C01840=1102.143,-108.620,-47.409,179.948,4.444,148.747
C01841=1102.137,-108.370,-47.419,179.947,4.449,148.749
C01842=1102.132,-108.121,-47.430,179.947,4.454,148.750
C01843=1102.128,-107.871,-47.440,179.946,4.459,148.751
C01844=1102.122,-107.621,-47.450,179.946,4.464,148.752
C01845=1102.117,-107.371,-47.460,179.946,4.469,148.753
C01846=1102.111,-107.122,-47.471,179.945,4.474,148.755
C01847=1102.106,-106.872,-47.481,179.944,4.479,148.756
C01848=1102.101,-106.622,-47.491,179.944,4.484,148.757
C01849=1102.096,-106.373,-47.501,179.944,4.489,148.758
C01850=1102.091,-106.122,-47.512,179.943,4.494,148.760
C01851=1102.085,-105.873,-47.522,179.943,4.499,148.761
C01852=1102.080,-105.623,-47.532,179.942,4.504,148.762
C01853=1102.075,-105.373,-47.543,179.942,4.509,148.763
C01854=1102.069,-105.124,-47.553,179.941,4.513,148.764
C01855=1102.064,-104.874,-47.564,179.941,4.518,148.766
C01856=1102.059,-104.624,-47.574,179.940,4.524,148.767
C01857=1102.054,-104.375,-47.584,179.940,4.529,148.768
C01858=1102.049,-104.125,-47.594,179.939,4.533,148.769
C01859=1102.043,-103.875,-47.605,179.939,4.539,148.771
C01860=1102.038,-103.625,-47.615,179.939,4.544,148.772
C01861=1102.033,-103.376,-47.625,179.938,4.548,148.773
C01862=1102.028,-103.126,-47.637,179.938,4.553,148.774
C01863=1102.023,-102.876,-47.647,179.938,4.558,148.775
C01864=1102.017,-102.627,-47.657,179.937,4.563,148.777
C01865=1102.012,-102.377,-47.668,179.937,4.568,148.778
C01866=1102.006,-102.127,-47.678,179.936,4.573,148.779
C01867=1102.001,-101.877,-47.689,179.936,4.578,148.780
C01868=1101.997,-101.628,-47.699,179.935,4.583,148.782
C01869=1101.992,-101.378,-47.709,179.935,4.588,148.783
C01870=1101.986,-101.128,-47.720,179.934,4.593,148.784
C01871=1101.981,-100.878,-47.730,179.933,4.597,148.785
C01872=1101.976,-100.664,-47.740,179.933,4.601,148.786
C01873=1101.972,-100.450,-47.748,179.933,4.606,148.787
C01874=1101.967,-100.235,-47.758,179.933,4.611,148.788
C01875=1101.963,-100.022,-47.767,179.932,4.614,148.789
C01876=1101.959,-99.806,-47.776,179.932,4.618,148.790
C01877=1101.954,-99.592,-47.785,179.931,4.623,148.792
C01878=1101.949,-99.378,-47.794,179.931,4.627,148.793
C01879=1101.944,-99.164,-47.803,179.931,4.631,148.793
C01880=1101.939,-98.913,-47.814,179.930,4.636,148.795
C01881=1101.934,-98.664,-47.825,179.930,4.641,148.796
C01882=1101.929,-98.414,-47.835,179.930,4.646,148.797
C01883=1101.923,-98.165,-47.845,179.929,4.651,148.799
C01884=1101.918,-97.914,-47.856,179.929,4.656,148.800
C01885=1101.913,-97.665,-47.867,179.928,4.661,148.801
C01886=1101.908,-97.415,-47.878,179.928,4.665,148.802
C01887=1101.903,-97.166,-47.888,179.927,4.671,148.803
C01888=1101.898,-96.916,-47.899,179.927,4.676,148.805
C01889=1101.892,-96.666,-47.909,179.926,4.680,148.806
C01890=1101.887,-96.416,-47.920,179.926,4.685,148.807
C01891=1101.882,-96.167,-47.931,179.926,4.690,148.808
C01892=1101.877,-95.917,-47.941,179.925,4.695,148.809
C01893=1101.872,-95.668,-47.952,179.925,4.700,148.810
C01894=1101.867,-95.418,-47.963,179.925,4.705,148.812
C01895=1101.862,-95.168,-47.973,179.924,4.709,148.813
C01896=1101.856,-94.919,-47.984,179.924,4.714,148.814
C01897=1101.851,-94.668,-47.995,179.923,4.720,148.815
C01898=1101.845,-94.419,-48.006,179.923,4.725,148.816
C01899=1101.840,-94.169,-48.017,179.922,4.729,148.818
C01900=1101.835,-93.919,-48.027,179.922,4.734,148.819
C01901=1101.830,-93.670,-48.038,179.922,4.739,148.820
C01902=1101.824,-93.420,-48.049,179.921,4.744,148.821
C01903=1101.820,-93.171,-48.060,179.921,4.749,148.822
C01904=1101.815,-92.920,-48.071,179.921,4.754,148.824
C01905=1101.809,-92.671,-48.082,179.921,4.759,148.825
C01906=1101.804,-92.421,-48.093,179.920,4.763,148.826
C01907=1101.798,-92.172,-48.104,179.920,4.769,148.827
C01908=1101.793,-91.922,-48.114,179.919,4.774,148.828
C01909=1101.788,-91.672,-48.125,179.919,4.779,148.830
C01910=1101.783,-91.423,-48.136,179.919,4.783,148.831
C01911=1101.778,-91.172,-48.146,179.918,4.788,148.832
C01912=1101.772,-90.923,-48.158,179.918,4.793,148.833
C01913=1101.767,-90.674,-48.169,179.918,4.799,148.834
C01914=1101.762,-90.423,-48.180,179.918,4.804,148.836
C01915=1101.757,-90.174,-48.191,179.917,4.808,148.837
C01916=1101.752,-89.924,-48.201,179.917,4.813,148.838
C01917=1101.747,-89.674,-48.213,179.917,4.818,148.839
C01918=1101.741,-89.425,-48.223,179.916,4.824,148.840
C01919=1101.736,-89.175,-48.234,179.916,4.829,148.841
C01920=1101.731,-88.925,-48.245,179.916,4.834,148.843
C01921=1101.726,-88.676,-48.256,179.915,4.838,148.844
C01922=1101.721,-88.426,-48.268,179.915,4.844,148.845
C01923=1101.715,-88.176,-48.278,179.914,4.849,148.846
C01924=1101.710,-87.927,-48.289,179.914,4.854,148.848
C01925=1101.705,-87.676,-48.300,179.914,4.859,148.849
C01926=1101.699,-87.427,-48.311,179.914,4.864,148.850
C01927=1101.695,-87.178,-48.323,179.913,4.869,148.851
C01928=1101.691,-86.964,-48.332,179.913,4.873,148.852
C01929=1101.686,-86.749,-48.342,179.913,4.878,148.853
C01930=1101.681,-86.535,-48.351,179.912,4.882,148.854
C01931=1101.677,-86.321,-48.360,179.913,4.886,148.855
C01932=1101.673,-86.106,-48.370,179.912,4.891,148.856
C01933=1101.668,-85.892,-48.380,179.912,4.895,148.857
C01934=1101.664,-85.678,-48.389,179.911,4.900,148.859
C01935=1101.659,-85.463,-48.399,179.911,4.904,148.860
C01936=1101.654,-85.214,-48.409,179.911,4.909,148.861
C01937=1101.649,-84.964,-48.421,179.911,4.914,148.862
C01938=1101.643,-84.714,-48.433,179.911,4.919,148.863
C01939=1101.638,-84.464,-48.443,179.910,4.923,148.864
C01940=1101.633,-84.215,-48.454,179.910,4.929,148.865
C01941=1101.628,-83.965,-48.466,179.909,4.934,148.867
C01942=1101.623,-83.715,-48.477,179.909,4.939,148.868
C01943=1101.617,-83.466,-48.487,179.909,4.944,148.869
C01944=1101.612,-83.216,-48.499,179.909,4.950,148.870
C01945=1101.607,-82.966,-48.511,179.908,4.955,148.872
C01946=1101.603,-82.717,-48.522,179.908,4.960,148.873
C01947=1101.596,-82.467,-48.533,179.908,4.965,148.874
C01948=1101.592,-82.217,-48.544,179.908,4.970,148.875
C01949=1101.586,-81.967,-48.556,179.907,4.974,148.876
C01950=1101.582,-81.718,-48.567,179.907,4.980,148.877
C01951=1101.576,-81.469,-48.578,179.906,4.985,148.879
C01952=1101.570,-81.218,-48.589,179.906,4.990,148.880
C01953=1101.566,-80.968,-48.601,179.906,4.995,148.881
C01954=1101.561,-80.719,-48.612,179.906,5.000,148.882
C01955=1101.555,-80.470,-48.623,179.906,5.006,148.884
C01956=1101.550,-80.220,-48.635,179.905,5.011,148.885
C01957=1101.545,-79.970,-48.647,179.905,5.016,148.886
C01958=1101.540,-79.720,-48.657,179.905,5.021,148.887
C01959=1101.534,-79.471,-48.669,179.905,5.026,148.888
C01960=1101.529,-79.221,-48.680,179.905,5.031,148.890
C01961=1101.524,-78.971,-48.692,179.905,5.036,148.891
C01962=1101.519,-78.721,-48.703,179.903,5.041,148.892
C01963=1101.514,-78.471,-48.715,179.903,5.046,148.893
C01964=1101.508,-78.223,-48.726,179.903,5.051,148.894
C01965=1101.504,-77.973,-48.737,179.903,5.057,148.896
C01966=1101.498,-77.723,-48.749,179.903,5.062,148.897
C01967=1101.493,-77.473,-48.760,179.903,5.067,148.898
C01968=1101.488,-77.223,-48.772,179.902,5.072,148.899
C01969=1101.483,-76.974,-48.782,179.902,5.077,148.900
C01970=1101.477,-76.724,-48.794,179.902,5.082,148.902
C01971=1101.472,-76.474,-48.806,179.902,5.087,148.903
C01972=1101.467,-76.224,-48.818,179.902,5.092,148.904
C01973=1101.462,-75.974,-48.829,179.902,5.098,148.905
C01974=1101.457,-75.725,-48.841,179.902,5.103,148.906
C01975=1101.451,-75.476,-48.852,179.901,5.108,148.907
C01976=1101.446,-75.226,-48.864,179.901,5.113,148.909
C01977=1101.441,-74.976,-48.875,179.901,5.118,148.910
C01978=1101.436,-74.726,-48.887,179.901,5.123,148.911
C01979=1101.431,-74.476,-48.899,179.901,5.128,148.912
C01980=1101.426,-74.227,-48.910,179.901,5.134,148.913
C01981=1101.420,-73.978,-48.921,179.900,5.138,148.914
C01982=1101.414,-73.728,-48.933,179.900,5.143,148.916
C01983=1101.410,-73.479,-48.945,179.900,5.148,148.917
C01984=1101.406,-73.264,-48.955,179.900,5.153,148.918
C01985=1101.401,-73.050,-48.965,179.899,5.157,148.919
C01986=1101.397,-72.835,-48.976,179.900,5.162,148.920
C01987=1101.392,-72.621,-48.985,179.899,5.166,148.921
C01988=1101.389,-72.407,-48.995,179.899,5.170,148.922
C01989=1101.384,-72.193,-49.005,179.899,5.175,148.923
C01990=1101.379,-71.979,-49.015,179.899,5.179,148.924
C01991=1101.375,-71.765,-49.025,179.899,5.183,148.925
C01992=1101.369,-71.515,-49.037,179.898,5.188,148.926
C01993=1101.365,-71.265,-49.049,179.898,5.193,148.927
C01994=1101.359,-71.015,-49.060,179.898,5.198,148.928
C01995=1101.354,-70.765,-49.072,179.898,5.203,148.929
C01996=1101.349,-70.516,-49.084,179.898,5.209,148.931
C01997=1101.343,-70.267,-49.096,179.898,5.214,148.932
C01998=1101.338,-70.017,-49.108,179.898,5.219,148.933
C01999=1101.333,-69.768,-49.119,179.898,5.224,148.934
C02000=1101.328,-69.518,-49.131,179.897,5.229,148.935
C02001=1101.322,-69.268,-49.143,179.898,5.234,148.936
C02002=1101.318,-69.019,-49.155,179.898,5.239,148.937
C02003=1101.312,-68.769,-49.167,179.898,5.244,148.939
C02004=1101.307,-68.519,-49.179,179.897,5.249,148.940
C02005=1101.302,-68.269,-49.190,179.897,5.254,148.941
C02006=1101.297,-68.020,-49.202,179.897,5.259,148.942
C02007=1101.292,-67.770,-49.214,179.897,5.265,148.943
C02008=1101.287,-67.520,-49.226,179.897,5.269,148.944
C02009=1101.282,-67.270,-49.238,179.897,5.274,148.945
C02010=1101.277,-67.021,-49.250,179.897,5.279,148.947
C02011=1101.271,-66.771,-49.262,179.896,5.284,148.948
C02012=1101.266,-66.521,-49.273,179.897,5.289,148.949
C02013=1101.261,-66.272,-49.286,179.897,5.294,148.950
C02014=1101.256,-66.022,-49.298,179.897,5.299,148.951
C02015=1101.250,-65.772,-49.310,179.896,5.304,148.952
C02016=1101.246,-65.523,-49.322,179.897,5.309,148.953
C02017=1101.241,-65.273,-49.334,179.897,5.314,148.954
C02018=1101.235,-65.023,-49.345,179.897,5.319,148.955
C02019=1101.230,-64.774,-49.358,179.896,5.324,148.957
C02020=1101.225,-64.524,-49.370,179.897,5.329,148.958
C02021=1101.220,-64.275,-49.381,179.897,5.334,148.959
C02022=1101.215,-64.025,-49.394,179.897,5.339,148.960
C02023=1101.209,-63.775,-49.406,179.897,5.344,148.961
C02024=1101.204,-63.526,-49.418,179.896,5.348,148.962
C02025=1101.199,-63.276,-49.430,179.897,5.353,148.963
C02026=1101.194,-63.026,-49.442,179.897,5.358,148.964
C02027=1101.189,-62.777,-49.454,179.896,5.363,148.965
C02028=1101.184,-62.527,-49.466,179.897,5.368,148.966
C02029=1101.178,-62.278,-49.479,179.897,5.373,148.967
C02030=1101.173,-62.028,-49.490,179.897,5.378,148.968
C02031=1101.168,-61.779,-49.503,179.897,5.383,148.969
C02032=1101.164,-61.528,-49.515,179.897,5.388,148.970
C02033=1101.159,-61.279,-49.527,179.897,5.393,148.971
C02034=1101.153,-61.029,-49.539,179.897,5.397,148.972
C02035=1101.148,-60.780,-49.552,179.897,5.402,148.974
C02036=1101.143,-60.530,-49.564,179.897,5.407,148.975
C02037=1101.138,-60.280,-49.576,179.897,5.412,148.976
C02038=1101.132,-60.030,-49.588,179.898,5.417,148.977
C02039=1101.127,-59.781,-49.601,179.898,5.422,148.978
C02040=1101.123,-59.567,-49.612,179.897,5.426,148.979
C02041=1101.118,-59.353,-49.621,179.897,5.430,148.980
C02042=1101.114,-59.139,-49.632,179.897,5.433,148.980
C02043=1101.110,-58.924,-49.643,179.898,5.438,148.981
C02044=1101.105,-58.711,-49.653,179.898,5.442,148.982
C02045=1101.101,-58.497,-49.664,179.897,5.446,148.983
C02046=1101.097,-58.282,-49.674,179.897,5.450,148.984
C02047=1101.092,-58.068,-49.684,179.897,5.454,148.985
C02048=1101.087,-57.819,-49.697,179.897,5.459,148.986
C02049=1101.083,-57.569,-49.710,179.897,5.464,148.987
C02050=1101.077,-57.319,-49.721,179.897,5.468,148.988
C02051=1101.072,-57.070,-49.734,179.897,5.473,148.989
C02052=1101.067,-56.820,-49.746,179.897,5.478,148.990
C02053=1101.062,-56.570,-49.759,179.896,5.482,148.991
C02054=1101.056,-56.321,-49.771,179.897,5.487,148.992
C02055=1101.051,-56.071,-49.783,179.897,5.492,148.994
C02056=1101.047,-55.821,-49.796,179.896,5.496,148.994
C02057=1101.041,-55.572,-49.809,179.896,5.501,148.996
C02058=1101.036,-55.322,-49.821,179.896,5.506,148.997
C02059=1101.031,-55.072,-49.833,179.896,5.510,148.998
C02060=1101.026,-54.823,-49.846,179.896,5.515,148.999
C02061=1101.020,-54.573,-49.858,179.896,5.520,149.000
C02062=1101.016,-54.323,-49.871,179.896,5.525,149.001
C02063=1101.011,-54.074,-49.883,179.896,5.529,149.002
C02064=1101.006,-53.825,-49.896,179.896,5.534,149.003
C02065=1101.000,-53.575,-49.908,179.896,5.539,149.004
C02066=1100.995,-53.325,-49.920,179.895,5.544,149.005
C02067=1100.990,-53.075,-49.933,179.896,5.548,149.006
C02068=1100.985,-52.826,-49.946,179.896,5.553,149.007
C02069=1100.980,-52.576,-49.958,179.895,5.558,149.009
C02070=1100.974,-52.326,-49.971,179.895,5.562,149.009
C02071=1100.969,-52.077,-49.983,179.895,5.568,149.011
C02072=1100.964,-51.827,-49.996,179.894,5.572,149.012
C02073=1100.959,-51.577,-50.008,179.895,5.577,149.013
C02074=1100.954,-51.328,-50.021,179.895,5.582,149.014
C02075=1100.949,-51.078,-50.034,179.894,5.586,149.015
C02076=1100.944,-50.828,-50.047,179.895,5.591,149.016
C02077=1100.939,-50.579,-50.059,179.894,5.596,149.017
C02078=1100.934,-50.329,-50.071,179.894,5.600,149.018
C02079=1100.929,-50.080,-50.084,179.894,5.605,149.019
C02080=1100.923,-49.830,-50.097,179.894,5.610,149.020
C02081=1100.918,-49.580,-50.110,179.893,5.614,149.022
C02082=1100.913,-49.331,-50.122,179.894,5.619,149.022
C02083=1100.908,-49.082,-50.135,179.894,5.624,149.024
C02084=1100.903,-48.832,-50.148,179.893,5.629,149.025
C02085=1100.898,-48.582,-50.160,179.894,5.633,149.026
C02086=1100.893,-48.332,-50.172,179.893,5.638,149.027
C02087=1100.887,-48.083,-50.186,179.893,5.643,149.028
C02088=1100.882,-47.833,-50.199,179.893,5.647,149.029
C02089=1100.877,-47.583,-50.211,179.893,5.652,149.030
C02090=1100.872,-47.334,-50.224,179.893,5.657,149.031
C02091=1100.867,-47.085,-50.236,179.892,5.662,149.032
C02092=1100.862,-46.834,-50.250,179.892,5.666,149.033
C02093=1100.857,-46.585,-50.263,179.892,5.671,149.034
C02094=1100.852,-46.336,-50.275,179.892,5.676,149.036
C02095=1100.847,-46.086,-50.288,179.892,5.680,149.036
C02096=1100.842,-45.872,-50.298,179.891,5.684,149.038
C02097=1100.838,-45.658,-50.310,179.892,5.689,149.039
C02098=1100.834,-45.443,-50.321,179.892,5.693,149.039
C02099=1100.829,-45.229,-50.333,179.891,5.697,149.040
C02100=1100.824,-45.016,-50.343,179.891,5.701,149.041
C02101=1100.820,-44.802,-50.354,179.891,5.705,149.042
C02102=1100.816,-44.587,-50.365,179.891,5.709,149.043
C02103=1100.812,-44.374,-50.376,179.891,5.713,149.044
C02104=1100.807,-44.124,-50.389,179.891,5.718,149.045
C02105=1100.801,-43.875,-50.402,179.891,5.723,149.046
C02106=1100.796,-43.625,-50.415,179.890,5.727,149.047
C02107=1100.791,-43.375,-50.428,179.890,5.732,149.048
C02108=1100.786,-43.126,-50.440,179.890,5.736,149.050
C02109=1100.781,-42.876,-50.454,179.890,5.741,149.051
C02110=1100.776,-42.626,-50.466,179.890,5.746,149.052
C02111=1100.771,-42.377,-50.479,179.889,5.751,149.053
C02112=1100.766,-42.127,-50.492,179.889,5.756,149.054
C02113=1100.760,-41.877,-50.505,179.890,5.760,149.055
C02114=1100.756,-41.627,-50.518,179.889,5.765,149.056
C02115=1100.751,-41.378,-50.531,179.890,5.769,149.057
C02116=1100.745,-41.128,-50.544,179.889,5.774,149.058
C02117=1100.740,-40.878,-50.557,179.889,5.779,149.059
C02118=1100.735,-40.630,-50.570,179.889,5.783,149.060
C02119=1100.730,-40.380,-50.583,179.889,5.788,149.061
C02120=1100.725,-40.130,-50.596,179.889,5.793,149.062
C02121=1100.720,-39.881,-50.609,179.889,5.797,149.063
C02122=1100.715,-39.630,-50.623,179.889,5.802,149.064
C02123=1100.710,-39.381,-50.635,179.889,5.806,149.065
C02124=1100.704,-39.131,-50.648,179.889,5.810,149.066
C02125=1100.700,-38.882,-50.662,179.889,5.816,149.067
C02126=1100.694,-38.633,-50.675,179.889,5.819,149.068
C02127=1100.689,-38.382,-50.688,179.889,5.824,149.069
C02128=1100.684,-38.133,-50.701,179.889,5.828,149.070
C02129=1100.679,-37.884,-50.713,179.890,5.833,149.071
C02130=1100.674,-37.634,-50.728,179.890,5.838,149.072
C02131=1100.669,-37.385,-50.740,179.890,5.842,149.073
C02132=1100.664,-37.134,-50.754,179.890,5.847,149.074
C02133=1100.658,-36.885,-50.767,179.890,5.851,149.075
C02134=1100.654,-36.636,-50.780,179.890,5.855,149.076
C02135=1100.648,-36.386,-50.793,179.890,5.859,149.077
C02136=1100.643,-36.137,-50.806,179.891,5.864,149.078
C02137=1100.638,-35.886,-50.820,179.891,5.869,149.078
C02138=1100.633,-35.638,-50.833,179.891,5.873,149.079
C02139=1100.628,-35.387,-50.846,179.891,5.877,149.080
C02140=1100.623,-35.138,-50.859,179.892,5.882,149.081
C02141=1100.618,-34.888,-50.873,179.892,5.886,149.082
C02142=1100.613,-34.639,-50.886,179.892,5.891,149.083
C02143=1100.607,-34.389,-50.899,179.892,5.895,149.084
C02144=1100.603,-34.140,-50.913,179.892,5.899,149.085
C02145=1100.598,-33.890,-50.926,179.893,5.904,149.086
C02146=1100.592,-33.640,-50.939,179.893,5.908,149.087
C02147=1100.588,-33.391,-50.953,179.893,5.913,149.088
C02148=1100.582,-33.141,-50.966,179.894,5.918,149.088
C02149=1100.578,-32.891,-50.979,179.893,5.921,149.089
C02150=1100.572,-32.642,-50.993,179.894,5.926,149.090
C02151=1100.568,-32.392,-51.006,179.895,5.931,149.091
C02152=1100.559,-32.014,-51.027,179.895,5.937,149.092
C02153=1100.552,-31.636,-51.047,179.896,5.944,149.094
C02154=1100.544,-31.258,-51.067,179.896,5.951,149.095
C02155=1100.536,-30.879,-51.087,179.896,5.957,149.096
C02156=1100.531,-30.629,-51.101,179.897,5.962,149.097
C02157=1100.526,-30.380,-51.114,179.897,5.967,149.098
C02158=1100.521,-30.130,-51.128,179.898,5.971,149.099
C02159=1100.515,-29.881,-51.141,179.898,5.975,149.100
C02160=1100.511,-29.631,-51.155,179.899,5.980,149.101
C02161=1100.505,-29.382,-51.168,179.899,5.984,149.102
C02162=1100.501,-29.132,-51.182,179.900,5.989,149.103
C02163=1100.495,-28.883,-51.195,179.900,5.994,149.103
C02164=1100.490,-28.633,-51.209,179.900,5.999,149.104
C02165=1100.486,-28.383,-51.222,179.900,6.003,149.105
C02166=1100.480,-28.134,-51.236,179.901,6.007,149.106
C02167=1100.476,-27.884,-51.249,179.901,6.012,149.107
C02168=1100.470,-27.635,-51.263,179.902,6.017,149.108
C02169=1100.465,-27.385,-51.277,179.902,6.021,149.109
C02170=1100.461,-27.135,-51.290,179.903,6.026,149.110
C02171=1100.455,-26.886,-51.304,179.903,6.031,149.111
C02172=1100.450,-26.636,-51.318,179.904,6.036,149.112
C02173=1100.445,-26.387,-51.331,179.904,6.040,149.113
C02174=1100.440,-26.138,-51.345,179.905,6.045,149.113
C02175=1100.435,-25.887,-51.359,179.905,6.050,149.114
C02176=1100.430,-25.638,-51.372,179.905,6.055,149.115
C02177=1100.425,-25.388,-51.386,179.906,6.059,149.116
C02178=1100.419,-25.139,-51.400,179.906,6.064,149.117
C02179=1100.415,-24.890,-51.413,179.906,6.068,149.118
C02180=1100.188,-34.518,-50.930,179.897,5.896,149.083
C02181=1100.194,-34.768,-50.916,179.897,5.892,149.082
C02182=1100.199,-35.018,-50.904,179.897,5.887,149.081
C02183=1100.204,-35.267,-50.890,179.897,5.882,149.080
C02184=1100.209,-35.517,-50.877,179.897,5.878,149.079
C02185=1100.214,-35.766,-50.864,179.896,5.874,149.078
C02186=1100.219,-36.016,-50.851,179.896,5.870,149.077
C02187=1100.224,-36.265,-50.837,179.896,5.865,149.076
C02188=1100.229,-36.515,-50.824,179.895,5.860,149.075
C02189=1100.234,-36.765,-50.811,179.896,5.856,149.074
C02190=1100.239,-37.014,-50.797,179.895,5.851,149.073
C02191=1100.244,-37.264,-50.784,179.895,5.848,149.072
C02192=1100.250,-37.514,-50.771,179.895,5.842,149.071
C02193=1100.255,-37.763,-50.758,179.896,5.838,149.070
C02194=1100.260,-38.012,-50.745,179.895,5.834,149.070
C02195=1100.265,-38.262,-50.731,179.895,5.829,149.069
C02196=1100.270,-38.512,-50.719,179.895,5.825,149.068
C02197=1100.275,-38.762,-50.705,179.895,5.820,149.067
C02198=1100.280,-39.011,-50.692,179.895,5.816,149.066
C02199=1100.285,-39.261,-50.679,179.895,5.811,149.065
C02200=1100.291,-39.510,-50.666,179.895,5.807,149.064
C02201=1100.296,-39.760,-50.653,179.895,5.802,149.063
C02202=1100.300,-40.010,-50.640,179.895,5.798,149.062
C02203=1100.306,-40.259,-50.627,179.895,5.793,149.061
C02204=1100.310,-40.509,-50.613,179.895,5.788,149.060
C02205=1100.316,-40.758,-50.600,179.895,5.784,149.059
C02206=1100.321,-41.008,-50.587,179.895,5.779,149.058
C02207=1100.326,-41.258,-50.574,179.895,5.775,149.056
C02208=1100.332,-41.507,-50.561,179.895,5.770,149.056
C02209=1100.337,-41.757,-50.549,179.896,5.766,149.054
C02210=1100.341,-42.007,-50.536,179.896,5.761,149.053
C02211=1100.347,-42.256,-50.522,179.895,5.756,149.052
C02212=1100.351,-42.506,-50.509,179.896,5.752,149.051
C02213=1100.356,-42.755,-50.496,179.896,5.747,149.050
C02214=1100.362,-43.004,-50.484,179.897,5.742,149.049
C02215=1100.367,-43.255,-50.470,179.896,5.738,149.048
C02216=1100.372,-43.504,-50.457,179.896,5.733,149.047
C02217=1100.377,-43.753,-50.445,179.897,5.728,149.046
C02218=1100.382,-44.004,-50.431,179.897,5.723,149.045
C02219=1100.387,-44.253,-50.419,179.896,5.718,149.044
C02220=1100.393,-44.502,-50.406,179.897,5.714,149.042
C02221=1100.400,-44.896,-50.386,179.897,5.706,149.041
C02222=1100.409,-45.290,-50.365,179.897,5.699,149.039
C02223=1100.416,-45.684,-50.345,179.898,5.692,149.037
C02224=1100.424,-46.077,-50.325,179.898,5.684,149.036
C02225=1100.430,-46.327,-50.312,179.898,5.679,149.034
C02226=1100.435,-46.577,-50.299,179.898,5.675,149.033
C02227=1100.440,-46.826,-50.286,179.898,5.670,149.032
C02228=1100.445,-47.076,-50.273,179.898,5.665,149.031
C02229=1100.450,-47.326,-50.260,179.899,5.661,149.030
C02230=1100.455,-47.575,-50.247,179.899,5.656,149.029
C02231=1100.460,-47.825,-50.235,179.899,5.651,149.028
C02232=1100.466,-48.075,-50.223,179.899,5.646,149.027
C02233=1100.470,-48.325,-50.210,179.899,5.642,149.026
C02234=1100.475,-48.574,-50.197,179.899,5.637,149.025
C02235=1100.481,-48.824,-50.184,179.900,5.632,149.024
C02236=1100.486,-49.074,-50.171,179.899,5.628,149.023
C02237=1100.491,-49.323,-50.158,179.899,5.622,149.021
C02238=1100.496,-49.572,-50.146,179.900,5.618,149.020
C02239=1100.501,-49.822,-50.133,179.900,5.613,149.019
C02240=1100.506,-50.072,-50.120,179.900,5.608,149.018
C02241=1100.512,-50.322,-50.108,179.900,5.604,149.017
C02242=1100.517,-50.571,-50.095,179.901,5.599,149.016
C02243=1100.522,-50.821,-50.083,179.900,5.594,149.015
C02244=1100.527,-51.071,-50.070,179.901,5.590,149.014
C02245=1100.532,-51.320,-50.057,179.901,5.585,149.013
C02246=1100.537,-51.569,-50.044,179.900,5.580,149.012
C02247=1100.542,-51.819,-50.033,179.901,5.576,149.011
C02248=1100.547,-52.068,-50.020,179.901,5.570,149.009
C02249=1100.552,-52.318,-50.007,179.901,5.566,149.009
C02250=1100.558,-52.568,-49.994,179.901,5.561,149.007
C02251=1100.563,-52.817,-49.981,179.902,5.556,149.006
C02252=1100.568,-53.067,-49.969,179.901,5.552,149.005
C02253=1100.573,-53.317,-49.956,179.902,5.547,149.004
C02254=1100.578,-53.567,-49.944,179.901,5.542,149.003
C02255=1100.583,-53.816,-49.931,179.901,5.537,149.002
C02256=1100.589,-54.066,-49.919,179.902,5.533,149.001
C02257=1100.594,-54.315,-49.907,179.902,5.528,149.000
C02258=1100.598,-54.565,-49.894,179.902,5.523,148.999
C02259=1100.603,-54.815,-49.881,179.903,5.519,148.998
C02260=1100.609,-55.064,-49.869,179.902,5.514,148.997
C02261=1100.614,-55.314,-49.857,179.902,5.509,148.996
C02262=1100.619,-55.563,-49.844,179.902,5.505,148.995
C02263=1100.624,-55.814,-49.832,179.903,5.500,148.994
C02264=1100.629,-56.063,-49.819,179.903,5.495,148.992
C02265=1100.634,-56.312,-49.807,179.903,5.491,148.991
C02266=1100.640,-56.562,-49.795,179.903,5.486,148.990
C02267=1100.645,-56.812,-49.782,179.902,5.481,148.989
C02268=1100.650,-57.061,-49.769,179.903,5.476,148.988
C02269=1100.655,-57.312,-49.757,179.903,5.472,148.987
C02270=1100.660,-57.561,-49.745,179.903,5.467,148.986
C02271=1100.665,-57.810,-49.732,179.903,5.462,148.985
C02272=1100.670,-58.060,-49.720,179.903,5.458,148.984
C02273=1100.674,-58.274,-49.709,179.903,5.454,148.983
C02274=1100.679,-58.488,-49.699,179.903,5.449,148.982
C02275=1100.683,-58.702,-49.688,179.903,5.445,148.981
C02276=1100.687,-58.916,-49.678,179.903,5.441,148.980
C02277=1100.692,-59.130,-49.667,179.904,5.437,148.979
C02278=1100.696,-59.345,-49.656,179.904,5.433,148.978
C02279=1100.701,-59.559,-49.646,179.904,5.429,148.978
C02280=1100.705,-59.773,-49.636,179.904,5.425,148.977
C02281=1100.710,-60.022,-49.623,179.903,5.420,148.976
C02282=1100.716,-60.272,-49.611,179.904,5.416,148.974
C02283=1100.721,-60.521,-49.599,179.903,5.411,148.974
C02284=1100.726,-60.771,-49.587,179.904,5.406,148.972
C02285=1100.730,-61.021,-49.574,179.903,5.401,148.971
C02286=1100.736,-61.271,-49.562,179.903,5.396,148.970
C02287=1100.741,-61.520,-49.550,179.903,5.391,148.969
C02288=1100.746,-61.770,-49.538,179.903,5.386,148.968
C02289=1100.751,-62.020,-49.525,179.903,5.381,148.967
C02290=1100.757,-62.270,-49.513,179.903,5.377,148.966
C02291=1100.762,-62.519,-49.501,179.903,5.372,148.965
C02292=1100.767,-62.768,-49.490,179.903,5.367,148.964
C02293=1100.772,-63.018,-49.477,179.903,5.362,148.963
C02294=1100.777,-63.268,-49.465,179.903,5.357,148.962
C02295=1100.782,-63.517,-49.452,179.903,5.352,148.961
C02296=1100.788,-63.767,-49.441,179.903,5.347,148.960
C02297=1100.793,-64.016,-49.428,179.903,5.342,148.959
C02298=1100.798,-64.266,-49.417,179.903,5.337,148.957
C02299=1100.803,-64.516,-49.405,179.903,5.333,148.957
C02300=1100.807,-64.766,-49.392,179.903,5.328,148.955
C02301=1100.813,-65.016,-49.380,179.903,5.323,148.954
C02302=1100.818,-65.265,-49.367,179.903,5.318,148.953
C02303=1100.823,-65.515,-49.356,179.903,5.313,148.952
C02304=1100.828,-65.765,-49.344,179.903,5.308,148.951
C02305=1100.833,-66.014,-49.332,179.903,5.303,148.950
C02306=1100.839,-66.264,-49.320,179.903,5.298,148.949
C02307=1100.843,-66.514,-49.308,179.903,5.293,148.948
C02308=1100.849,-66.763,-49.296,179.903,5.288,148.947
C02309=1100.854,-67.013,-49.284,179.903,5.283,148.945
C02310=1100.859,-67.263,-49.272,179.903,5.277,148.944
C02311=1100.864,-67.512,-49.260,179.903,5.273,148.943
C02312=1100.869,-67.762,-49.248,179.904,5.268,148.942
C02313=1100.875,-68.012,-49.236,179.904,5.263,148.941
C02314=1100.880,-68.262,-49.224,179.904,5.258,148.940
C02315=1100.884,-68.511,-49.212,179.904,5.253,148.939
C02316=1100.890,-68.761,-49.200,179.904,5.248,148.937
C02317=1100.896,-69.010,-49.189,179.904,5.243,148.936
C02318=1100.901,-69.259,-49.178,179.904,5.238,148.935
C02319=1100.906,-69.509,-49.165,179.904,5.233,148.934
C02320=1100.911,-69.759,-49.153,179.904,5.228,148.933
C02321=1100.917,-70.009,-49.141,179.904,5.223,148.932
C02322=1100.921,-70.258,-49.130,179.904,5.217,148.931
C02323=1100.927,-70.508,-49.118,179.905,5.212,148.929
C02324=1100.932,-70.757,-49.105,179.905,5.207,148.928
C02325=1100.937,-71.007,-49.094,179.905,5.202,148.927
C02326=1100.942,-71.257,-49.082,179.905,5.197,148.926
C02327=1100.947,-71.507,-49.070,179.905,5.192,148.925
C02328=1100.952,-71.757,-49.059,179.905,5.187,148.924
C02329=1100.957,-71.970,-49.049,179.905,5.183,148.923
C02330=1100.961,-72.185,-49.039,179.906,5.179,148.922
C02331=1100.966,-72.399,-49.028,179.905,5.174,148.921
C02332=1100.970,-72.613,-49.018,179.906,5.170,148.920
C02333=1100.975,-72.827,-49.008,179.906,5.166,148.919
C02334=1100.978,-73.041,-48.999,179.906,5.161,148.918
C02335=1100.983,-73.256,-48.989,179.906,5.157,148.917
C02336=1100.987,-73.470,-48.978,179.906,5.152,148.916
C02337=1100.993,-73.719,-48.967,179.906,5.147,148.914
C02338=1100.998,-73.969,-48.955,179.907,5.142,148.913
C02339=1101.003,-74.219,-48.944,179.907,5.137,148.912
C02340=1101.009,-74.469,-48.932,179.907,5.132,148.911
C02341=1101.013,-74.718,-48.920,179.908,5.127,148.910
C02342=1101.019,-74.968,-48.909,179.908,5.122,148.909
C02343=1101.024,-75.218,-48.897,179.908,5.117,148.907
C02344=1101.030,-75.467,-48.886,179.908,5.112,148.906
C02345=1101.034,-75.717,-48.874,179.908,5.107,148.905
C02346=1101.040,-75.967,-48.863,179.908,5.101,148.904
C02347=1101.044,-76.216,-48.851,179.908,5.096,148.903
C02348=1101.050,-76.466,-48.839,179.909,5.091,148.902
C02349=1101.055,-76.716,-48.827,179.909,5.086,148.900
C02350=1101.060,-76.966,-48.816,179.909,5.081,148.899
C02351=1101.066,-77.215,-48.805,179.909,5.076,148.898
C02352=1101.071,-77.465,-48.793,179.909,5.071,148.897
C02353=1101.076,-77.715,-48.781,179.909,5.065,148.896
C02354=1101.081,-77.964,-48.770,179.910,5.060,148.894
C02355=1101.086,-78.214,-48.758,179.910,5.055,148.893
C02356=1101.092,-78.463,-48.747,179.910,5.051,148.892
C02357=1101.097,-78.713,-48.736,179.911,5.046,148.891
C02358=1101.102,-78.963,-48.724,179.911,5.041,148.890
C02359=1101.107,-79.212,-48.712,179.911,5.035,148.888
C02360=1101.112,-79.462,-48.701,179.912,5.030,148.887
C02361=1101.117,-79.711,-48.690,179.912,5.025,148.886
C02362=1101.123,-79.961,-48.678,179.912,5.020,148.885
C02363=1101.128,-80.211,-48.668,179.912,5.014,148.884
C02364=1101.133,-80.461,-48.656,179.912,5.009,148.882
C02365=1101.138,-80.711,-48.644,179.912,5.004,148.881
C02366=1101.144,-80.960,-48.633,179.913,4.999,148.880
C02367=1101.148,-81.210,-48.622,179.913,4.994,148.879
C02368=1101.154,-81.460,-48.610,179.913,4.989,148.878
C02369=1101.158,-81.709,-48.599,179.914,4.984,148.876
C02370=1101.164,-81.959,-48.588,179.914,4.979,148.875
C02371=1101.170,-82.209,-48.576,179.914,4.974,148.874
C02372=1101.174,-82.458,-48.565,179.915,4.969,148.873
C02373=1101.180,-82.708,-48.553,179.915,4.964,148.872
C02374=1101.185,-82.957,-48.542,179.915,4.958,148.870
C02375=1101.190,-83.207,-48.532,179.915,4.953,148.869
C02376=1101.195,-83.457,-48.520,179.915,4.948,148.868
C02377=1101.200,-83.707,-48.509,179.915,4.943,148.867
C02378=1101.205,-83.956,-48.498,179.916,4.938,148.866
C02379=1101.211,-84.206,-48.486,179.916,4.932,148.864
C02380=1101.216,-84.456,-48.475,179.917,4.928,148.863
C02381=1101.221,-84.705,-48.464,179.917,4.923,148.862
C02382=1101.226,-84.955,-48.452,179.917,4.918,148.861
C02383=1101.231,-85.205,-48.442,179.918,4.913,148.859
C02384=1101.236,-85.455,-48.431,179.918,4.907,148.858
C02385=1101.241,-85.669,-48.421,179.918,4.904,148.857
C02386=1101.246,-85.883,-48.411,179.918,4.898,148.856
C02387=1101.250,-86.098,-48.402,179.919,4.894,148.855
C02388=1101.255,-86.312,-48.392,179.919,4.890,148.854
C02389=1101.259,-86.526,-48.383,179.919,4.885,148.853
C02390=1101.263,-86.741,-48.373,179.919,4.881,148.852
C02391=1101.268,-86.955,-48.363,179.920,4.877,148.851
C02392=1101.272,-87.169,-48.354,179.920,4.872,148.850
C02393=1101.278,-87.418,-48.343,179.920,4.868,148.849
C02394=1101.282,-87.668,-48.331,179.921,4.863,148.848
C02395=1101.288,-87.918,-48.321,179.921,4.858,148.846
C02396=1101.293,-88.167,-48.310,179.921,4.853,148.845
C02397=1101.298,-88.417,-48.298,179.921,4.847,148.844
C02398=1101.304,-88.667,-48.288,179.921,4.842,148.843
C02399=1101.308,-88.916,-48.276,179.923,4.838,148.841
C02400=1101.313,-89.167,-48.266,179.923,4.832,148.840
C02401=1101.319,-89.416,-48.254,179.923,4.827,148.839
C02402=1101.324,-89.665,-48.243,179.923,4.822,148.838
C02403=1101.329,-89.916,-48.232,179.923,4.817,148.837
C02404=1101.334,-90.165,-48.222,179.924,4.812,148.836
C02405=1101.339,-90.415,-48.211,179.924,4.808,148.834
C02406=1101.345,-90.664,-48.199,179.925,4.802,148.833
C02407=1101.350,-90.914,-48.189,179.925,4.797,148.832
C02408=1101.355,-91.164,-48.178,179.925,4.792,148.831
C02409=1101.361,-91.414,-48.167,179.925,4.787,148.830
C02410=1101.365,-91.663,-48.156,179.926,4.783,148.828
C02411=1101.371,-91.914,-48.145,179.926,4.777,148.827
C02412=1101.376,-92.163,-48.134,179.926,4.772,148.826
C02413=1101.381,-92.413,-48.123,179.927,4.767,148.825
C02414=1101.387,-92.662,-48.112,179.927,4.763,148.824
C02415=1101.392,-92.912,-48.102,179.927,4.758,148.822
C02416=1101.396,-93.162,-48.091,179.928,4.753,148.821
C02417=1101.402,-93.411,-48.080,179.928,4.747,148.820
C02418=1101.407,-93.661,-48.068,179.929,4.743,148.819
C02419=1101.413,-93.911,-48.058,179.929,4.738,148.818
C02420=1101.418,-94.160,-48.047,179.929,4.733,148.816
C02421=1101.423,-94.410,-48.037,179.929,4.728,148.815
C02422=1101.428,-94.659,-48.025,179.930,4.723,148.814
C02423=1101.433,-94.910,-48.015,179.930,4.718,148.813
C02424=1101.439,-95.159,-48.005,179.930,4.713,148.812
C02425=1101.443,-95.409,-47.993,179.931,4.709,148.810
C02426=1101.450,-95.659,-47.983,179.931,4.704,148.809
C02427=1101.454,-95.908,-47.971,179.932,4.698,148.808
C02428=1101.460,-96.158,-47.961,179.932,4.694,148.807
C02429=1101.465,-96.408,-47.951,179.933,4.689,148.806
C02430=1101.470,-96.657,-47.940,179.933,4.684,148.804
C02431=1101.475,-96.907,-47.929,179.934,4.680,148.803
C02432=1101.480,-97.157,-47.918,179.934,4.674,148.802
C02433=1101.486,-97.407,-47.908,179.934,4.669,148.801
C02434=1101.491,-97.657,-47.897,179.935,4.665,148.800
C02435=1101.496,-97.906,-47.886,179.935,4.660,148.799
C02436=1101.501,-98.156,-47.875,179.935,4.655,148.797
C02437=1101.506,-98.405,-47.865,179.936,4.650,148.796
C02438=1101.511,-98.655,-47.854,179.936,4.645,148.795
C02439=1101.517,-98.905,-47.844,179.937,4.640,148.794
C02440=1101.522,-99.155,-47.833,179.937,4.636,148.793
C02441=1101.527,-99.369,-47.824,179.938,4.631,148.791
C02442=1101.531,-99.584,-47.815,179.938,4.627,148.790
C02443=1101.536,-99.798,-47.806,179.938,4.623,148.789
C02444=1101.540,-100.011,-47.797,179.939,4.618,148.788
C02445=1101.544,-100.227,-47.788,179.939,4.614,148.787
C02446=1101.549,-100.441,-47.778,179.940,4.610,148.786
C02447=1101.553,-100.655,-47.769,179.940,4.605,148.785
C02448=1101.559,-100.869,-47.760,179.940,4.601,148.784
C02449=1101.564,-101.120,-47.750,179.941,4.597,148.783
C02450=1101.569,-101.369,-47.739,179.941,4.592,148.782
C02451=1101.574,-101.619,-47.728,179.941,4.587,148.781
C02452=1101.579,-101.868,-47.718,179.942,4.582,148.779
C02453=1101.584,-102.119,-47.707,179.943,4.577,148.778
C02454=1101.589,-102.367,-47.697,179.943,4.572,148.777
C02455=1101.594,-102.618,-47.686,179.943,4.566,148.775
C02456=1101.600,-102.867,-47.676,179.944,4.562,148.774
C02457=1101.605,-103.117,-47.666,179.944,4.557,148.773
C02458=1101.610,-103.367,-47.655,179.945,4.552,148.772
C02459=1101.615,-103.616,-47.645,179.945,4.548,148.771
C02460=1101.620,-103.866,-47.634,179.946,4.542,148.769
C02461=1101.626,-104.116,-47.624,179.946,4.537,148.768
C02462=1101.631,-104.366,-47.613,179.947,4.533,148.767
C02463=1101.637,-104.615,-47.603,179.947,4.528,148.766
C02464=1101.642,-104.866,-47.592,179.948,4.522,148.764
C02465=1101.647,-105.115,-47.582,179.948,4.517,148.763
C02466=1101.652,-105.364,-47.572,179.949,4.513,148.762
C02467=1101.657,-105.614,-47.561,179.949,4.508,148.761
C02468=1101.662,-105.864,-47.551,179.949,4.502,148.760
C02469=1101.667,-106.114,-47.541,179.950,4.498,148.758
C02470=1101.673,-106.363,-47.530,179.950,4.493,148.757
C02471=1101.679,-106.613,-47.520,179.951,4.488,148.756
C02472=1101.684,-106.863,-47.510,179.951,4.483,148.755
C02473=1101.689,-107.113,-47.499,179.952,4.478,148.753
C02474=1101.693,-107.363,-47.489,179.952,4.473,148.752
C02475=1101.699,-107.612,-47.479,179.953,4.468,148.751
C02476=1101.705,-107.862,-47.469,179.953,4.463,148.750
C02477=1101.710,-108.112,-47.458,179.954,4.458,148.749
C02478=1101.715,-108.361,-47.448,179.954,4.453,148.747
C02479=1101.720,-108.611,-47.437,179.955,4.448,148.746
C02480=1101.725,-108.860,-47.427,179.955,4.443,148.745
C02481=1101.730,-109.110,-47.417,179.956,4.438,148.743
C02482=1101.735,-109.360,-47.406,179.956,4.433,148.742
C02483=1101.741,-109.610,-47.396,179.956,4.428,148.741
C02484=1101.747,-109.859,-47.386,179.957,4.423,148.740
C02485=1101.751,-110.109,-47.376,179.958,4.418,148.738
C02486=1101.756,-110.359,-47.366,179.958,4.413,148.737
C02487=1101.762,-110.609,-47.356,179.958,4.408,148.736
C02488=1101.767,-110.859,-47.346,179.959,4.403,148.735
C02489=1101.773,-111.109,-47.336,179.959,4.398,148.734
C02490=1101.778,-111.358,-47.326,179.960,4.393,148.732
C02491=1101.783,-111.608,-47.315,179.960,4.387,148.731
C02492=1101.788,-111.858,-47.305,179.961,4.383,148.730
C02493=1101.794,-112.107,-47.295,179.962,4.378,148.728
C02494=1101.798,-112.357,-47.285,179.962,4.373,148.727
C02495=1101.804,-112.607,-47.275,179.963,4.367,148.726
C02496=1101.809,-112.856,-47.265,179.963,4.363,148.725
C02497=1101.814,-113.071,-47.256,179.963,4.358,148.724
C02498=1101.818,-113.286,-47.248,179.964,4.354,148.722
C02499=1101.822,-113.500,-47.239,179.964,4.350,148.721
C02500=1101.827,-113.714,-47.230,179.965,4.346,148.720
C02501=1101.832,-113.929,-47.221,179.965,4.341,148.719
C02502=1101.836,-114.143,-47.213,179.966,4.336,148.718
C02503=1101.841,-114.357,-47.204,179.966,4.332,148.717
C02504=1101.845,-114.572,-47.196,179.967,4.328,148.716
C02505=1101.851,-114.821,-47.185,179.967,4.323,148.715
C02506=1101.856,-115.071,-47.175,179.968,4.317,148.713
C02507=1101.861,-115.321,-47.166,179.968,4.312,148.712
C02508=1101.866,-115.571,-47.156,179.969,4.308,148.711
C02509=1101.872,-115.820,-47.145,179.969,4.303,148.710
C02510=1101.876,-116.070,-47.135,179.970,4.297,148.708
C02511=1101.882,-116.320,-47.125,179.970,4.292,148.707
C02512=1101.887,-116.569,-47.115,179.971,4.287,148.706
C02513=1101.893,-116.819,-47.106,179.972,4.282,148.704
C02514=1101.898,-117.070,-47.096,179.972,4.277,148.703
C02515=1101.903,-117.319,-47.085,179.973,4.272,148.702
C02516=1101.908,-117.568,-47.076,179.973,4.266,148.700
C02517=1101.914,-117.818,-47.066,179.974,4.261,148.699
C02518=1101.919,-118.069,-47.056,179.974,4.256,148.698
C02519=1101.924,-118.318,-47.046,179.975,4.251,148.696
C02520=1101.929,-118.567,-47.036,179.976,4.246,148.695
C02521=1101.935,-118.818,-47.026,179.976,4.241,148.694
C02522=1101.940,-119.068,-47.016,179.977,4.236,148.692
C02523=1101.945,-119.317,-47.006,179.977,4.230,148.691
C02524=1101.950,-119.566,-46.997,179.978,4.226,148.690
C02525=1101.956,-119.817,-46.987,179.979,4.221,148.689
C02526=1101.962,-120.066,-46.977,179.979,4.215,148.687
C02527=1101.966,-120.316,-46.967,179.980,4.210,148.686
C02528=1101.972,-120.566,-46.957,179.980,4.205,148.685
C02529=1101.977,-120.815,-46.948,179.981,4.199,148.683
C02530=1101.982,-121.065,-46.938,179.981,4.194,148.682
C02531=1101.987,-121.315,-46.929,179.982,4.190,148.681
C02532=1101.992,-121.565,-46.918,179.983,4.184,148.679
C02533=1101.997,-121.814,-46.909,179.983,4.179,148.678
C02534=1102.003,-122.064,-46.899,179.984,4.173,148.677
C02535=1102.009,-122.314,-46.889,179.984,4.168,148.675
C02536=1102.014,-122.564,-46.880,179.985,4.163,148.674
C02537=1102.019,-122.814,-46.869,179.985,4.158,148.673
C02538=1102.024,-123.063,-46.860,179.986,4.153,148.671
C02539=1102.030,-123.313,-46.850,179.987,4.148,148.670
C02540=1102.035,-123.563,-46.841,179.988,4.142,148.669
C02541=1102.040,-123.812,-46.830,179.988,4.137,148.667
C02542=1102.045,-124.062,-46.822,179.989,4.132,148.666
C02543=1102.050,-124.312,-46.811,179.989,4.126,148.665
C02544=1102.055,-124.562,-46.802,179.990,4.121,148.663
C02545=1102.061,-124.812,-46.792,179.990,4.116,148.662
C02546=1102.066,-125.062,-46.783,179.991,4.111,148.661
C02547=1102.072,-125.311,-46.773,179.992,4.106,148.659
C02548=1102.077,-125.561,-46.764,179.993,4.100,148.658
C02549=1102.083,-125.811,-46.754,179.993,4.095,148.657
C02550=1102.088,-126.060,-46.745,179.994,4.090,148.655
C02551=1102.092,-126.310,-46.735,179.994,4.084,148.654
C02552=1102.098,-126.560,-46.725,179.995,4.079,148.652
C02553=1102.102,-126.775,-46.717,179.996,4.075,148.651
C02554=1102.107,-126.989,-46.709,179.996,4.069,148.650
C02555=1102.111,-127.204,-46.700,179.996,4.065,148.649
C02556=1102.116,-127.418,-46.692,179.997,4.061,148.648
C02557=1102.121,-127.632,-46.684,179.998,4.056,148.647
C02558=1102.126,-127.847,-46.676,179.998,4.052,148.645
C02559=1102.130,-128.061,-46.667,179.999,4.046,148.644
C02560=1102.134,-128.276,-46.660,180.000,4.042,148.643
C02561=1101.711,-128.266,-46.686,-179.993,4.047,148.642
C02562=1101.706,-128.052,-46.694,-179.994,4.051,148.643
C02563=1101.702,-127.838,-46.702,-179.994,4.056,148.644
C02564=1101.698,-127.624,-46.710,-179.995,4.060,148.645
C02565=1101.693,-127.409,-46.718,-179.996,4.065,148.646
C02566=1101.688,-127.194,-46.726,-179.996,4.070,148.648
C02567=1101.684,-126.980,-46.734,-179.997,4.074,148.649
C02568=1101.679,-126.765,-46.743,-179.998,4.078,148.650
C02569=1101.675,-126.551,-46.751,-179.998,4.084,148.651
C02570=1101.669,-126.301,-46.761,-179.998,4.089,148.652
C02571=1101.664,-126.051,-46.770,-179.999,4.094,148.654
C02572=1101.659,-125.801,-46.781,-180.000,4.099,148.655
C02573=1101.654,-125.551,-46.789,179.999,4.104,148.657
C02574=1101.648,-125.302,-46.800,179.999,4.109,148.658
C02575=1101.644,-125.052,-46.809,179.998,4.115,148.659
C02576=1101.638,-124.802,-46.819,179.998,4.120,148.661
C02577=1101.633,-124.553,-46.828,179.997,4.126,148.662
C02578=1101.627,-124.303,-46.838,179.996,4.131,148.663
C02579=1101.623,-124.053,-46.848,179.996,4.136,148.665
C02580=1101.617,-123.803,-46.857,179.995,4.142,148.666
C02581=1101.612,-123.553,-46.867,179.994,4.146,148.667
C02582=1101.606,-123.304,-46.877,179.993,4.152,148.669
C02583=1101.601,-123.054,-46.886,179.993,4.157,148.670
C02584=1101.595,-122.805,-46.896,179.992,4.162,148.672
C02585=1101.591,-122.555,-46.906,179.992,4.167,148.673
C02586=1101.585,-122.304,-46.916,179.992,4.173,148.674
C02587=1101.580,-122.055,-46.925,179.991,4.178,148.675
C02588=1101.575,-121.806,-46.936,179.990,4.182,148.677
C02589=1101.569,-121.555,-46.945,179.989,4.188,148.678
C02590=1101.565,-121.306,-46.955,179.989,4.193,148.679
C02591=1101.559,-121.056,-46.965,179.988,4.199,148.681
C02592=1101.554,-120.806,-46.974,179.988,4.204,148.682
C02593=1101.548,-120.557,-46.984,179.987,4.209,148.683
C02594=1101.543,-120.306,-46.995,179.986,4.214,148.685
C02595=1101.538,-120.057,-47.004,179.986,4.219,148.686
C02596=1101.533,-119.807,-47.014,179.985,4.224,148.687
C02597=1101.528,-119.558,-47.024,179.985,4.230,148.689
C02598=1101.522,-119.308,-47.034,179.984,4.235,148.690
C02599=1101.517,-119.057,-47.044,179.984,4.240,148.691
C02600=1101.512,-118.808,-47.053,179.983,4.245,148.692
C02601=1101.506,-118.559,-47.064,179.982,4.250,148.694
C02602=1101.501,-118.309,-47.073,179.982,4.255,148.695
C02603=1101.496,-118.058,-47.083,179.982,4.260,148.696
C02604=1101.491,-117.809,-47.093,179.981,4.266,148.698
C02605=1101.486,-117.560,-47.103,179.980,4.270,148.699
C02606=1101.480,-117.310,-47.113,179.980,4.275,148.700
C02607=1101.475,-117.060,-47.124,179.979,4.281,148.702
C02608=1101.470,-116.810,-47.132,179.979,4.286,148.703
C02609=1101.464,-116.560,-47.143,179.978,4.291,148.704
C02610=1101.459,-116.311,-47.153,179.977,4.296,148.706
C02611=1101.454,-116.061,-47.163,179.977,4.301,148.707
C02612=1101.449,-115.811,-47.173,179.976,4.306,148.708
C02613=1101.443,-115.562,-47.183,179.976,4.312,148.710
C02614=1101.438,-115.311,-47.193,179.975,4.317,148.711
C02615=1101.433,-115.062,-47.203,179.975,4.321,148.712
C02616=1101.428,-114.812,-47.213,179.974,4.327,148.713
C02617=1101.422,-114.563,-47.223,179.973,4.332,148.715
C02618=1101.418,-114.348,-47.232,179.973,4.336,148.716
C02619=1101.414,-114.134,-47.241,179.972,4.340,148.717
C02620=1101.409,-113.919,-47.249,179.973,4.345,148.718
C02621=1101.405,-113.705,-47.258,179.972,4.349,148.719
C02622=1101.400,-113.490,-47.267,179.971,4.353,148.720
C02623=1101.395,-113.276,-47.276,179.971,4.358,148.721
C02624=1101.391,-113.062,-47.284,179.970,4.363,148.722
C02625=1101.386,-112.847,-47.292,179.970,4.367,148.723
C02626=1101.381,-112.598,-47.302,179.970,4.372,148.725
C02627=1101.376,-112.347,-47.313,179.969,4.376,148.726
C02628=1101.370,-112.098,-47.323,179.968,4.382,148.727
C02629=1101.365,-111.849,-47.333,179.968,4.387,148.728
C02630=1101.360,-111.598,-47.343,179.968,4.392,148.730
C02631=1101.355,-111.349,-47.354,179.967,4.396,148.731
C02632=1101.349,-111.099,-47.364,179.966,4.402,148.732
C02633=1101.345,-110.849,-47.374,179.966,4.407,148.734
C02634=1101.339,-110.600,-47.384,179.966,4.412,148.735
C02635=1101.334,-110.350,-47.394,179.965,4.417,148.736
C02636=1101.329,-110.100,-47.405,179.964,4.422,148.737
C02637=1101.323,-109.851,-47.415,179.964,4.427,148.739
C02638=1101.319,-109.601,-47.425,179.963,4.432,148.740
C02639=1101.313,-109.351,-47.435,179.963,4.437,148.741
C02640=1101.308,-109.102,-47.445,179.962,4.442,148.742
C02641=1101.303,-108.851,-47.456,179.962,4.447,148.743
C02642=1101.297,-108.602,-47.466,179.961,4.451,148.745
C02643=1101.291,-108.352,-47.476,179.961,4.457,148.746
C02644=1101.286,-108.102,-47.487,179.960,4.462,148.747
C02645=1101.282,-107.853,-47.497,179.960,4.467,148.749
C02646=1101.277,-107.603,-47.508,179.959,4.471,148.750
C02647=1101.271,-107.354,-47.518,179.959,4.477,148.751
C02648=1101.266,-107.104,-47.528,179.959,4.482,148.752
C02649=1101.261,-106.854,-47.539,179.957,4.486,148.754
C02650=1101.255,-106.604,-47.549,179.957,4.492,148.755
C02651=1101.250,-106.354,-47.560,179.957,4.497,148.756
C02652=1101.245,-106.105,-47.569,179.957,4.502,148.757
C02653=1101.240,-105.855,-47.580,179.956,4.506,148.758
C02654=1101.235,-105.605,-47.590,179.956,4.511,148.760
C02655=1101.229,-105.356,-47.601,179.955,4.517,148.761
C02656=1101.224,-105.106,-47.612,179.955,4.521,148.762
C02657=1101.219,-104.856,-47.622,179.954,4.526,148.763
C02658=1101.214,-104.606,-47.632,179.954,4.532,148.765
C02659=1101.208,-104.356,-47.643,179.953,4.537,148.766
C02660=1101.203,-104.106,-47.653,179.953,4.541,148.767
C02661=1101.198,-103.857,-47.664,179.952,4.546,148.768
C02662=1101.193,-103.607,-47.675,179.952,4.551,148.769
C02663=1101.187,-103.358,-47.685,179.951,4.556,148.771
C02664=1101.182,-103.107,-47.695,179.951,4.561,148.772
C02665=1101.177,-102.858,-47.705,179.951,4.566,148.773
C02666=1101.172,-102.609,-47.716,179.950,4.570,148.774
C02667=1101.167,-102.359,-47.726,179.950,4.575,148.775
C02668=1101.162,-102.109,-47.737,179.949,4.581,148.777
C02669=1101.157,-101.859,-47.747,179.949,4.586,148.778
C02670=1101.151,-101.610,-47.758,179.948,4.590,148.779
C02671=1101.146,-101.360,-47.769,179.948,4.596,148.781
C02672=1101.141,-101.110,-47.779,179.948,4.601,148.782
C02673=1101.136,-100.860,-47.790,179.947,4.605,148.783
C02674=1101.131,-100.646,-47.799,179.946,4.609,148.784
C02675=1101.126,-100.432,-47.808,179.946,4.614,148.785
C02676=1101.122,-100.218,-47.817,179.946,4.618,148.786
C02677=1101.118,-100.003,-47.827,179.946,4.622,148.787
C02678=1101.113,-99.789,-47.836,179.945,4.626,148.788
C02679=1101.108,-99.574,-47.845,179.945,4.630,148.789
C02680=1101.104,-99.360,-47.854,179.944,4.634,148.790
C02681=1101.099,-99.146,-47.863,179.944,4.639,148.791
C02682=1101.094,-98.896,-47.874,179.943,4.644,148.793
C02683=1101.088,-98.646,-47.884,179.943,4.649,148.794
C02684=1101.084,-98.397,-47.895,179.943,4.654,148.795
C02685=1101.078,-98.147,-47.905,179.942,4.658,148.796
C02686=1101.073,-97.897,-47.916,179.942,4.664,148.797
C02687=1101.068,-97.647,-47.927,179.942,4.669,148.799
C02688=1101.063,-97.398,-47.938,179.941,4.673,148.800
C02689=1101.058,-97.148,-47.948,179.941,4.678,148.801
C02690=1101.053,-96.899,-47.959,179.940,4.683,148.802
C02691=1101.048,-96.648,-47.970,179.940,4.688,148.803
C02692=1101.042,-96.399,-47.981,179.939,4.693,148.804
C02693=1101.037,-96.149,-47.991,179.939,4.698,148.806
C02694=1101.031,-95.899,-48.002,179.938,4.702,148.807
C02695=1101.026,-95.650,-48.013,179.938,4.707,148.808
C02696=1101.021,-95.400,-48.023,179.938,4.713,148.809
C02697=1101.016,-95.151,-48.035,179.937,4.717,148.810
C02698=1101.011,-94.900,-48.045,179.937,4.722,148.812
C02699=1101.006,-94.651,-48.056,179.937,4.727,148.813
C02700=1101.001,-94.401,-48.067,179.936,4.731,148.814
C02701=1100.995,-94.152,-48.078,179.936,4.737,148.815
C02702=1100.990,-93.902,-48.089,179.936,4.742,148.816
C02703=1100.985,-93.652,-48.100,179.935,4.746,148.818
C02704=1100.979,-93.403,-48.110,179.935,4.751,148.819
C02705=1100.975,-93.153,-48.122,179.934,4.756,148.820
C02706=1100.969,-92.903,-48.132,179.934,4.762,148.821
C02707=1100.964,-92.654,-48.143,179.934,4.767,148.822
C02708=1100.959,-92.403,-48.154,179.933,4.771,148.824
C02709=1100.953,-92.154,-48.165,179.933,4.776,148.825
C02710=1100.948,-91.904,-48.176,179.933,4.781,148.826
C02711=1100.943,-91.655,-48.187,179.933,4.786,148.827
C02712=1100.938,-91.405,-48.197,179.932,4.791,148.828
C02713=1100.933,-91.155,-48.209,179.932,4.796,148.830
C02714=1100.927,-90.905,-48.219,179.931,4.801,148.831
C02715=1100.922,-90.656,-48.231,179.931,4.806,148.832
C02716=1100.917,-90.405,-48.241,179.931,4.811,148.833
C02717=1100.912,-90.157,-48.252,179.931,4.816,148.834
C02718=1100.907,-89.907,-48.264,179.930,4.821,148.835
C02719=1100.902,-89.656,-48.275,179.930,4.826,148.837
C02720=1100.896,-89.407,-48.286,179.930,4.831,148.838
C02721=1100.891,-89.157,-48.296,179.929,4.836,148.839
C02722=1100.886,-88.907,-48.308,179.929,4.842,148.840
C02723=1100.881,-88.658,-48.319,179.928,4.846,148.842
C02724=1100.876,-88.408,-48.330,179.928,4.851,148.843
C02725=1100.871,-88.158,-48.341,179.928,4.856,148.844
C02726=1100.865,-87.909,-48.352,179.927,4.861,148.845
C02727=1100.860,-87.659,-48.363,179.927,4.867,148.846
C02728=1100.855,-87.409,-48.374,179.927,4.872,148.848
C02729=1100.849,-87.160,-48.386,179.927,4.877,148.849
C02730=1100.846,-86.946,-48.395,179.927,4.881,148.850
C02731=1100.841,-86.731,-48.405,179.926,4.885,148.851
C02732=1100.836,-86.518,-48.414,179.926,4.890,148.852
C02733=1100.832,-86.303,-48.424,179.925,4.894,148.853
C02734=1100.827,-86.089,-48.434,179.925,4.898,148.854
C02735=1100.823,-85.875,-48.443,179.925,4.903,148.855
C02736=1100.819,-85.660,-48.453,179.925,4.907,148.856
C02737=1100.814,-85.446,-48.462,179.924,4.911,148.857
C02738=1100.809,-85.196,-48.473,179.924,4.916,148.858
C02739=1100.804,-84.947,-48.484,179.924,4.922,148.859
C02740=1100.798,-84.697,-48.496,179.924,4.927,148.861
C02741=1100.793,-84.447,-48.507,179.924,4.932,148.862
C02742=1100.789,-84.197,-48.518,179.924,4.937,148.863
C02743=1100.783,-83.948,-48.530,179.922,4.942,148.864
C02744=1100.778,-83.699,-48.541,179.922,4.947,148.866
C02745=1100.773,-83.448,-48.552,179.922,4.952,148.867
C02746=1100.767,-83.198,-48.563,179.922,4.957,148.868
C02747=1100.762,-82.949,-48.574,179.922,4.962,148.869
C02748=1100.757,-82.699,-48.586,179.921,4.967,148.870
C02749=1100.752,-82.450,-48.598,179.921,4.972,148.872
C02750=1100.747,-82.200,-48.608,179.921,4.978,148.873
C02751=1100.741,-81.950,-48.620,179.921,4.983,148.874
C02752=1100.736,-81.701,-48.631,179.920,4.988,148.875
C02753=1100.731,-81.451,-48.643,179.920,4.993,148.877
C02754=1100.726,-81.201,-48.654,179.919,4.998,148.878
C02755=1100.722,-80.952,-48.665,179.919,5.003,148.879
C02756=1100.715,-80.702,-48.677,179.919,5.008,148.880
C02757=1100.711,-80.453,-48.688,179.919,5.013,148.881
C02758=1100.705,-80.202,-48.699,179.919,5.018,148.882
C02759=1100.700,-79.952,-48.711,179.919,5.023,148.884
C02760=1100.695,-79.703,-48.723,179.918,5.029,148.885
C02761=1100.690,-79.454,-48.733,179.918,5.034,148.886
C02762=1100.684,-79.204,-48.745,179.918,5.039,148.887
C02763=1100.680,-78.954,-48.757,179.917,5.044,148.889
C02764=1100.674,-78.704,-48.769,179.917,5.049,148.890
C02765=1100.669,-78.455,-48.780,179.917,5.055,148.891
C02766=1100.663,-78.205,-48.791,179.917,5.060,148.892
C02767=1100.659,-77.956,-48.803,179.917,5.065,148.893
C02768=1100.653,-77.706,-48.815,179.916,5.069,148.894
C02769=1100.649,-77.456,-48.826,179.916,5.074,148.896
C02770=1100.643,-77.206,-48.838,179.916,5.079,148.897
C02771=1100.638,-76.957,-48.849,179.916,5.085,148.898
C02772=1100.632,-76.707,-48.860,179.915,5.090,148.899
C02773=1100.627,-76.457,-48.872,179.915,5.095,148.900
C02774=1100.622,-76.208,-48.884,179.915,5.100,148.902
C02775=1100.617,-75.958,-48.896,179.915,5.105,148.903
C02776=1100.612,-75.708,-48.907,179.915,5.110,148.904
C02777=1100.607,-75.458,-48.919,179.915,5.115,148.905
C02778=1100.602,-75.209,-48.930,179.915,5.121,148.906
C02779=1100.596,-74.959,-48.942,179.914,5.126,148.908
C02780=1100.591,-74.709,-48.953,179.914,5.131,148.909
C02781=1100.586,-74.460,-48.965,179.914,5.136,148.910
C02782=1100.580,-74.210,-48.977,179.913,5.141,148.911
C02783=1100.576,-73.961,-48.989,179.913,5.147,148.912
C02784=1100.571,-73.711,-49.000,179.913,5.152,148.914
C02785=1100.565,-73.461,-49.012,179.912,5.156,148.915
C02786=1100.561,-73.247,-49.021,179.913,5.161,148.916
C02787=1100.557,-73.033,-49.032,179.913,5.165,148.917
C02788=1100.552,-72.819,-49.042,179.913,5.169,148.917
C02789=1100.548,-72.605,-49.052,179.912,5.174,148.919
C02790=1100.543,-72.390,-49.062,179.912,5.178,148.920
C02791=1100.538,-72.177,-49.072,179.912,5.182,148.921
C02792=1100.534,-71.962,-49.082,179.912,5.186,148.921
C02793=1100.529,-71.748,-49.092,179.911,5.191,148.923
C02794=1100.525,-71.499,-49.104,179.911,5.196,148.924
C02795=1100.519,-71.249,-49.116,179.911,5.201,148.925
C02796=1100.514,-70.999,-49.128,179.911,5.206,148.926
C02797=1100.509,-70.749,-49.139,179.911,5.211,148.927
C02798=1100.504,-70.500,-49.152,179.911,5.216,148.928
C02799=1100.499,-70.250,-49.164,179.911,5.221,148.929
C02800=1100.494,-70.000,-49.175,179.911,5.226,148.931
C02801=1100.489,-69.751,-49.187,179.911,5.231,148.932
C02802=1100.483,-69.501,-49.199,179.911,5.237,148.933
C02803=1100.479,-69.252,-49.211,179.911,5.242,148.934
C02804=1100.473,-69.002,-49.223,179.910,5.247,148.935
C02805=1100.468,-68.752,-49.235,179.910,5.252,148.936
C02806=1100.463,-68.502,-49.247,179.911,5.257,148.937
C02807=1100.458,-68.253,-49.258,179.910,5.262,148.939
C02808=1100.453,-68.003,-49.270,179.910,5.266,148.940
C02809=1100.447,-67.753,-49.282,179.910,5.271,148.941
C02810=1100.442,-67.504,-49.295,179.910,5.276,148.942
C02811=1100.437,-67.254,-49.306,179.909,5.282,148.943
C02812=1100.432,-67.004,-49.318,179.910,5.286,148.944
C02813=1100.427,-66.755,-49.331,179.910,5.291,148.945
C02814=1100.421,-66.505,-49.342,179.910,5.297,148.947
C02815=1100.417,-66.255,-49.354,179.909,5.302,148.948
C02816=1100.412,-66.006,-49.366,179.909,5.307,148.949
C02817=1100.406,-65.756,-49.378,179.910,5.312,148.950
C02818=1100.401,-65.507,-49.391,179.910,5.317,148.951
C02819=1100.396,-65.257,-49.403,179.909,5.322,148.952
C02820=1100.391,-65.007,-49.414,179.909,5.326,148.953
C02821=1100.386,-64.758,-49.427,179.909,5.331,148.954
C02822=1100.380,-64.508,-49.438,179.909,5.336,148.955
C02823=1100.375,-64.258,-49.451,179.909,5.341,148.957
C02824=1100.370,-64.008,-49.463,179.909,5.346,148.957
C02825=1100.365,-63.759,-49.476,179.909,5.351,148.959
C02826=1100.360,-63.510,-49.487,179.909,5.356,148.960
C02827=1100.355,-63.260,-49.499,179.909,5.361,148.961
C02828=1100.349,-63.010,-49.511,179.909,5.366,148.962
C02829=1100.345,-62.760,-49.524,179.909,5.370,148.963
C02830=1100.340,-62.510,-49.536,179.909,5.375,148.964
C02831=1100.334,-62.260,-49.548,179.909,5.380,148.965
C02832=1100.329,-62.011,-49.561,179.909,5.385,148.966
C02833=1100.324,-61.761,-49.572,179.909,5.390,148.967
C02834=1100.319,-61.512,-49.585,179.910,5.395,148.968
C02835=1100.314,-61.262,-49.596,179.909,5.400,148.969
C02836=1100.309,-61.013,-49.609,179.910,5.405,148.970
C02837=1100.303,-60.764,-49.622,179.909,5.409,148.971
C02838=1100.298,-60.514,-49.634,179.910,5.414,148.972
C02839=1100.294,-60.264,-49.647,179.909,5.419,148.974
C02840=1100.288,-60.014,-49.658,179.910,5.424,148.974
C02841=1100.283,-59.764,-49.671,179.910,5.429,148.976
C02842=1100.278,-59.551,-49.681,179.909,5.433,148.977
C02843=1100.274,-59.337,-49.692,179.909,5.437,148.977
C02844=1100.270,-59.122,-49.702,179.909,5.441,148.978
C02845=1100.265,-58.908,-49.712,179.910,5.445,148.979
C02846=1100.261,-58.694,-49.723,179.910,5.449,148.980
C02847=1100.257,-58.480,-49.734,179.910,5.453,148.981
C02848=1100.252,-58.266,-49.745,179.909,5.457,148.982
C02849=1100.248,-58.052,-49.756,179.909,5.461,148.983
C02850=1100.243,-57.802,-49.768,179.909,5.466,148.984
C02851=1100.237,-57.552,-49.780,179.909,5.471,148.985
C02852=1100.232,-57.303,-49.793,179.909,5.475,148.986
C02853=1100.227,-57.054,-49.805,179.909,5.480,148.987
C02854=1100.222,-56.803,-49.817,179.909,5.485,148.988
C02855=1100.217,-56.554,-49.830,179.908,5.489,148.989
C02856=1100.212,-56.304,-49.843,179.909,5.494,148.990
C02857=1100.207,-56.055,-49.855,179.909,5.499,148.991
C02858=1100.201,-55.805,-49.867,179.909,5.503,148.992
C02859=1100.197,-55.555,-49.880,179.908,5.508,148.994
C02860=1100.192,-55.306,-49.893,179.908,5.513,148.995
C02861=1100.186,-55.056,-49.905,179.908,5.517,148.996
C02862=1100.181,-54.807,-49.917,179.908,5.522,148.997
C02863=1100.176,-54.557,-49.930,179.908,5.527,148.998
C02864=1100.172,-54.307,-49.943,179.908,5.532,148.999
C02865=1100.166,-54.057,-49.955,179.908,5.536,149.000
C02866=1100.161,-53.808,-49.967,179.908,5.541,149.001
C02867=1100.156,-53.559,-49.980,179.908,5.546,149.002
C02868=1100.151,-53.309,-49.992,179.907,5.551,149.003
C02869=1100.146,-53.059,-50.005,179.908,5.555,149.004
C02870=1100.141,-52.809,-50.017,179.908,5.560,149.005
C02871=1100.136,-52.560,-50.030,179.907,5.565,149.006
C02872=1100.131,-52.311,-50.043,179.907,5.569,149.007
C02873=1100.125,-52.060,-50.056,179.907,5.575,149.009
C02874=1100.120,-51.811,-50.068,179.907,5.579,149.010
C02875=1100.115,-51.561,-50.081,179.907,5.584,149.011
C02876=1100.110,-51.312,-50.093,179.907,5.589,149.012
C02877=1100.105,-51.062,-50.106,179.906,5.593,149.013
C02878=1100.100,-50.813,-50.119,179.907,5.598,149.014
C02879=1100.095,-50.563,-50.131,179.907,5.603,149.015
C02880=1100.089,-50.314,-50.145,179.906,5.607,149.016
C02881=1100.084,-50.063,-50.157,179.906,5.612,149.017
C02882=1100.079,-49.814,-50.169,179.906,5.617,149.018
C02883=1100.074,-49.564,-50.182,179.906,5.621,149.019
C02884=1100.069,-49.315,-50.195,179.906,5.626,149.020
C02885=1100.064,-49.065,-50.208,179.906,5.631,149.021
C02886=1100.058,-48.815,-50.221,179.905,5.636,149.023
C02887=1100.053,-48.566,-50.233,179.906,5.640,149.024
C02888=1100.049,-48.316,-50.246,179.906,5.645,149.025
C02889=1100.044,-48.067,-50.259,179.905,5.650,149.026
C02890=1100.039,-47.817,-50.272,179.905,5.655,149.027
C02891=1100.033,-47.568,-50.285,179.905,5.660,149.028
C02892=1100.028,-47.318,-50.298,179.905,5.664,149.029
C02893=1100.023,-47.068,-50.310,179.905,5.669,149.030
C02894=1100.018,-46.819,-50.323,179.905,5.674,149.031
C02895=1100.013,-46.569,-50.336,179.904,5.678,149.032
C02896=1100.008,-46.319,-50.349,179.904,5.683,149.033
C02897=1100.002,-46.070,-50.362,179.904,5.687,149.034
C02898=1099.997,-45.824,-50.374,179.904,5.692,149.036
C02899=1099.992,-45.578,-50.387,179.904,5.697,149.037
C02900=1099.988,-45.333,-50.400,179.904,5.701,149.038
C02901=1099.983,-45.087,-50.412,179.904,5.706,149.039
C02902=1099.977,-44.841,-50.425,179.903,5.711,149.040
C02903=1099.973,-44.595,-50.438,179.904,5.715,149.041
C02904=1099.967,-44.350,-50.450,179.903,5.721,149.042
C02905=1099.962,-44.103,-50.463,179.903,5.725,149.043
C02906=1099.736,-53.659,-50.011,179.913,5.547,149.001
C02907=1099.742,-53.909,-49.997,179.914,5.543,149.000
C02908=1099.746,-54.159,-49.985,179.914,5.538,148.998
C02909=1099.751,-54.408,-49.972,179.914,5.533,148.997
C02910=1099.757,-54.658,-49.960,179.914,5.529,148.996
C02911=1099.762,-54.908,-49.947,179.914,5.524,148.995
C02912=1099.766,-55.158,-49.934,179.914,5.519,148.994
C02913=1099.772,-55.407,-49.922,179.915,5.514,148.993
C02914=1099.777,-55.657,-49.910,179.914,5.510,148.992
C02915=1099.782,-55.906,-49.897,179.914,5.505,148.991
C02916=1099.787,-56.156,-49.885,179.915,5.500,148.990
C02917=1099.792,-56.406,-49.873,179.915,5.496,148.989
C02918=1099.797,-56.655,-49.860,179.915,5.490,148.988
C02919=1099.802,-56.905,-49.847,179.915,5.486,148.987
C02920=1099.807,-57.154,-49.835,179.915,5.481,148.986
C02921=1099.813,-57.404,-49.823,179.915,5.476,148.984
C02922=1099.818,-57.653,-49.810,179.915,5.471,148.984
C02923=1099.823,-57.903,-49.797,179.916,5.467,148.982
C02924=1099.828,-58.153,-49.785,179.915,5.462,148.981
C02925=1099.833,-58.403,-49.773,179.915,5.457,148.980
C02926=1099.838,-58.652,-49.760,179.915,5.453,148.979
C02927=1099.844,-58.928,-49.747,179.916,5.448,148.978
C02928=1099.850,-59.204,-49.733,179.916,5.442,148.977
C02929=1099.855,-59.480,-49.720,179.916,5.437,148.976
C02930=1099.861,-59.756,-49.706,179.916,5.432,148.974
C02931=1099.866,-60.005,-49.693,179.915,5.427,148.974
C02932=1099.871,-60.256,-49.681,179.916,5.423,148.972
C02933=1099.876,-60.505,-49.668,179.916,5.418,148.971
C02934=1099.881,-60.755,-49.657,179.916,5.413,148.970
C02935=1099.886,-61.004,-49.644,179.915,5.408,148.969
C02936=1099.891,-61.254,-49.632,179.915,5.403,148.968
C02937=1099.897,-61.504,-49.620,179.915,5.398,148.967
C02938=1099.902,-61.753,-49.607,179.916,5.394,148.966
C02939=1099.907,-62.003,-49.595,179.915,5.389,148.965
C02940=1099.912,-62.253,-49.583,179.915,5.384,148.964
C02941=1099.917,-62.503,-49.571,179.915,5.379,148.963
C02942=1099.922,-62.752,-49.558,179.915,5.374,148.962
C02943=1099.928,-63.002,-49.546,179.915,5.369,148.961
C02944=1099.932,-63.251,-49.534,179.915,5.364,148.960
C02945=1099.938,-63.501,-49.522,179.915,5.359,148.959
C02946=1099.943,-63.750,-49.510,179.916,5.355,148.957
C02947=1099.948,-64.000,-49.498,179.915,5.350,148.957
C02948=1099.953,-64.250,-49.485,179.915,5.345,148.955
C02949=1099.959,-64.499,-49.473,179.916,5.340,148.954
C02950=1099.963,-64.748,-49.461,179.915,5.335,148.953
C02951=1099.969,-64.998,-49.449,179.915,5.330,148.952
C02952=1099.974,-65.248,-49.438,179.915,5.325,148.951
C02953=1099.978,-65.498,-49.425,179.916,5.320,148.950
C02954=1099.984,-65.748,-49.413,179.916,5.316,148.949
C02955=1099.989,-65.998,-49.400,179.916,5.311,148.948
C02956=1099.994,-66.247,-49.389,179.916,5.305,148.947
C02957=1099.999,-66.497,-49.377,179.916,5.300,148.945
C02958=1100.004,-66.747,-49.364,179.916,5.296,148.944
C02959=1100.010,-66.996,-49.352,179.916,5.290,148.943
C02960=1100.015,-67.246,-49.340,179.916,5.285,148.942
C02961=1100.020,-67.495,-49.328,179.916,5.280,148.941
C02962=1100.025,-67.745,-49.317,179.916,5.275,148.940
C02963=1100.030,-67.995,-49.304,179.916,5.270,148.939
C02964=1100.036,-68.245,-49.292,179.916,5.265,148.938
C02965=1100.040,-68.494,-49.281,179.917,5.261,148.936
C02966=1100.045,-68.744,-49.268,179.917,5.256,148.935
C02967=1100.051,-68.993,-49.256,179.917,5.251,148.934
C02968=1100.056,-69.243,-49.244,179.917,5.245,148.933
C02969=1100.061,-69.493,-49.233,179.917,5.240,148.932
C02970=1100.066,-69.742,-49.221,179.917,5.235,148.931
C02971=1100.071,-69.992,-49.209,179.918,5.230,148.929
C02972=1100.076,-70.242,-49.197,179.917,5.225,148.928
C02973=1100.082,-70.492,-49.186,179.917,5.220,148.927
C02974=1100.087,-70.741,-49.173,179.917,5.215,148.926
C02975=1100.092,-70.991,-49.161,179.918,5.210,148.925
C02976=1100.097,-71.240,-49.150,179.918,5.205,148.924
C02977=1100.103,-71.490,-49.138,179.918,5.200,148.923
C02978=1100.108,-71.739,-49.126,179.918,5.195,148.921
C02979=1100.112,-71.954,-49.116,179.918,5.191,148.921
C02980=1100.116,-72.167,-49.106,179.919,5.186,148.919
C02981=1100.121,-72.382,-49.096,179.919,5.182,148.918
C02982=1100.125,-72.596,-49.085,179.919,5.178,148.917
C02983=1100.129,-72.811,-49.075,179.919,5.174,148.917
C02984=1100.134,-73.024,-49.065,179.919,5.168,148.915
C02985=1100.138,-73.239,-49.055,179.919,5.165,148.914
C02986=1100.143,-73.453,-49.045,179.919,5.160,148.913
C02987=1100.148,-73.702,-49.033,179.920,5.155,148.912
C02988=1100.153,-73.952,-49.022,179.920,5.150,148.911
C02989=1100.159,-74.202,-49.010,179.920,5.145,148.910
C02990=1100.163,-74.452,-48.998,179.920,5.140,148.909
C02991=1100.169,-74.702,-48.987,179.920,5.135,148.908
C02992=1100.174,-74.951,-48.976,179.920,5.130,148.906
C02993=1100.179,-75.200,-48.963,179.921,5.125,148.905
C02994=1100.185,-75.450,-48.951,179.921,5.120,148.904
C02995=1100.189,-75.699,-48.940,179.921,5.114,148.903
C02996=1100.195,-75.949,-48.928,179.922,5.109,148.902
C02997=1100.199,-76.199,-48.917,179.922,5.104,148.900
C02998=1100.205,-76.449,-48.905,179.922,5.099,148.899
C02999=1100.210,-76.699,-48.893,179.922,5.093,148.898
C03000=1100.216,-76.948,-48.882,179.922,5.088,148.897
C03001=1100.221,-77.198,-48.870,179.922,5.083,148.896
C03002=1100.226,-77.447,-48.859,179.923,5.079,148.894
C03003=1100.231,-77.697,-48.847,179.923,5.074,148.893
C03004=1100.236,-77.947,-48.836,179.923,5.069,148.892
C03005=1100.241,-78.197,-48.824,179.924,5.063,148.891
C03006=1100.247,-78.446,-48.813,179.924,5.058,148.890
C03007=1100.252,-78.696,-48.801,179.924,5.053,148.889
C03008=1100.257,-78.945,-48.790,179.924,5.048,148.887
C03009=1100.262,-79.195,-48.778,179.924,5.043,148.886
C03010=1100.267,-79.445,-48.766,179.925,5.037,148.885
C03011=1100.272,-79.695,-48.755,179.925,5.032,148.884
C03012=1100.277,-79.944,-48.744,179.925,5.027,148.882
C03013=1100.283,-80.194,-48.732,179.925,5.022,148.881
C03014=1100.288,-80.443,-48.720,179.925,5.017,148.880
C03015=1100.293,-80.693,-48.709,179.926,5.012,148.879
C03016=1100.298,-80.943,-48.698,179.926,5.007,148.878
C03017=1100.304,-81.193,-48.686,179.927,5.002,148.877
C03018=1100.309,-81.442,-48.675,179.927,4.997,148.875
C03019=1100.314,-81.692,-48.663,179.927,4.992,148.874
C03020=1100.319,-81.942,-48.652,179.928,4.987,148.873
C03021=1100.324,-82.192,-48.640,179.928,4.981,148.872
C03022=1100.330,-82.441,-48.629,179.928,4.976,148.870
C03023=1100.334,-82.690,-48.618,179.928,4.971,148.869
C03024=1100.340,-82.941,-48.607,179.928,4.966,148.868
C03025=1100.345,-83.191,-48.595,179.928,4.961,148.867
C03026=1100.351,-83.440,-48.584,179.929,4.956,148.866
C03027=1100.355,-83.689,-48.573,179.929,4.951,148.864
C03028=1100.360,-83.939,-48.561,179.929,4.946,148.863
C03029=1100.366,-84.189,-48.549,179.930,4.941,148.862
C03030=1100.371,-84.439,-48.539,179.930,4.936,148.861
C03031=1100.377,-84.688,-48.527,179.931,4.930,148.859
C03032=1100.381,-84.938,-48.516,179.931,4.925,148.858
C03033=1100.386,-85.188,-48.505,179.931,4.920,148.857
C03034=1100.392,-85.438,-48.494,179.931,4.915,148.856
C03035=1100.396,-85.651,-48.484,179.931,4.911,148.855
C03036=1100.401,-85.866,-48.474,179.932,4.907,148.854
C03037=1100.405,-86.080,-48.465,179.932,4.902,148.853
C03038=1100.409,-86.294,-48.455,179.932,4.898,148.852
C03039=1100.414,-86.508,-48.446,179.933,4.894,148.851
C03040=1100.418,-86.722,-48.437,179.932,4.889,148.850
C03041=1100.423,-86.937,-48.427,179.933,4.885,148.849
C03042=1100.427,-87.151,-48.417,179.933,4.881,148.848
C03043=1100.432,-87.401,-48.406,179.934,4.876,148.846
C03044=1100.437,-87.650,-48.395,179.934,4.870,148.845
C03045=1100.443,-87.900,-48.383,179.934,4.865,148.844
C03046=1100.448,-88.150,-48.372,179.934,4.860,148.843
C03047=1100.453,-88.399,-48.361,179.934,4.855,148.842
C03048=1100.458,-88.649,-48.351,179.935,4.851,148.840
C03049=1100.464,-88.899,-48.339,179.935,4.846,148.839
C03050=1100.468,-89.149,-48.328,179.936,4.840,148.838
C03051=1100.474,-89.398,-48.317,179.936,4.835,148.837
C03052=1100.479,-89.648,-48.306,179.936,4.830,148.835
C03053=1100.484,-89.898,-48.294,179.937,4.825,148.834
C03054=1100.490,-90.147,-48.284,179.937,4.820,148.833
C03055=1100.494,-90.397,-48.273,179.938,4.815,148.832
C03056=1100.499,-90.647,-48.262,179.938,4.810,148.831
C03057=1100.505,-90.897,-48.251,179.938,4.805,148.830
C03058=1100.510,-91.146,-48.239,179.938,4.800,148.828
C03059=1100.516,-91.396,-48.229,179.938,4.795,148.827
C03060=1100.520,-91.645,-48.218,179.939,4.790,148.826
C03061=1100.526,-91.896,-48.207,179.939,4.785,148.825
C03062=1100.531,-92.145,-48.196,179.940,4.780,148.824
C03063=1100.536,-92.395,-48.185,179.940,4.775,148.822
C03064=1100.541,-92.645,-48.174,179.941,4.770,148.821
C03065=1100.546,-92.894,-48.163,179.941,4.765,148.820
C03066=1100.551,-93.144,-48.152,179.941,4.760,148.819
C03067=1100.557,-93.393,-48.141,179.941,4.755,148.818
C03068=1100.562,-93.643,-48.130,179.941,4.750,148.816
C03069=1100.567,-93.893,-48.119,179.942,4.746,148.815
C03070=1100.573,-94.143,-48.109,179.942,4.740,148.814
C03071=1100.577,-94.392,-48.097,179.943,4.735,148.813
C03072=1100.583,-94.643,-48.086,179.943,4.731,148.812
C03073=1100.588,-94.892,-48.075,179.944,4.726,148.810
C03074=1100.593,-95.142,-48.065,179.944,4.721,148.809
C03075=1100.599,-95.391,-48.055,179.945,4.716,148.808
C03076=1100.604,-95.641,-48.043,179.945,4.711,148.807
C03077=1100.609,-95.891,-48.033,179.945,4.706,148.806
C03078=1100.614,-96.140,-48.022,179.946,4.702,148.804
C03079=1100.619,-96.390,-48.011,179.946,4.697,148.803
C03080=1100.625,-96.640,-48.000,179.946,4.691,148.802
C03081=1100.630,-96.890,-47.989,179.947,4.687,148.801
C03082=1100.636,-97.139,-47.979,179.947,4.682,148.800
C03083=1100.640,-97.389,-47.968,179.947,4.677,148.798
C03084=1100.646,-97.639,-47.957,179.948,4.672,148.797
C03085=1100.651,-97.888,-47.946,179.948,4.667,148.796
C03086=1100.656,-98.138,-47.936,179.949,4.662,148.795
C03087=1100.661,-98.388,-47.925,179.949,4.658,148.794
C03088=1100.666,-98.638,-47.914,179.950,4.653,148.793
C03089=1100.671,-98.887,-47.904,179.950,4.648,148.791
C03090=1100.676,-99.137,-47.893,179.951,4.643,148.790
C03091=1100.681,-99.352,-47.884,179.951,4.638,148.789
C03092=1100.686,-99.565,-47.875,179.951,4.634,148.788
C03093=1100.691,-99.780,-47.865,179.951,4.630,148.787
C03094=1100.695,-99.994,-47.857,179.952,4.626,148.786
C03095=1100.699,-100.209,-47.847,179.953,4.622,148.785
C03096=1100.704,-100.423,-47.838,179.953,4.618,148.784
C03097=1100.708,-100.637,-47.829,179.953,4.613,148.783
C03098=1100.713,-100.851,-47.820,179.953,4.609,148.782
C03099=1100.718,-101.102,-47.809,179.954,4.605,148.781
C03100=1100.723,-101.351,-47.798,179.954,4.599,148.779
C03101=1100.728,-101.601,-47.787,179.955,4.594,148.778
C03102=1100.734,-101.850,-47.777,179.955,4.590,148.777
C03103=1100.739,-102.100,-47.766,179.956,4.585,148.776
C03104=1100.744,-102.350,-47.756,179.956,4.580,148.775
C03105=1100.749,-102.600,-47.745,179.957,4.574,148.773
C03106=1100.755,-102.849,-47.735,179.957,4.570,148.772
C03107=1100.759,-103.099,-47.724,179.958,4.565,148.771
C03108=1100.765,-103.348,-47.714,179.958,4.559,148.769
C03109=1100.771,-103.598,-47.703,179.959,4.555,148.768
C03110=1100.776,-103.848,-47.693,179.959,4.550,148.767
C03111=1100.781,-104.098,-47.683,179.959,4.545,148.766
C03112=1100.785,-104.347,-47.672,179.960,4.541,148.765
C03113=1100.791,-104.597,-47.662,179.960,4.535,148.763
C03114=1100.796,-104.847,-47.651,179.960,4.530,148.762
C03115=1100.801,-105.096,-47.641,179.962,4.526,148.761
C03116=1100.806,-105.347,-47.630,179.962,4.520,148.760
C03117=1100.812,-105.596,-47.619,179.962,4.515,148.758
C03118=1100.817,-105.846,-47.609,179.962,4.510,148.757
C03119=1100.822,-106.095,-47.599,179.963,4.506,148.756
C03120=1100.828,-106.345,-47.588,179.964,4.501,148.755
C03121=1100.833,-106.595,-47.578,179.964,4.495,148.754
C03122=1100.838,-106.845,-47.568,179.965,4.491,148.752
C03123=1100.843,-107.095,-47.557,179.965,4.486,148.751
C03124=1100.848,-107.344,-47.547,179.966,4.480,148.750
C03125=1100.853,-107.594,-47.536,179.966,4.475,148.749
C03126=1100.859,-107.843,-47.526,179.967,4.471,148.747
C03127=1100.864,-108.093,-47.516,179.967,4.466,148.746
C03128=1100.869,-108.343,-47.505,179.967,4.461,148.745
C03129=1100.875,-108.593,-47.495,179.968,4.456,148.743
C03130=1100.880,-108.843,-47.484,179.969,4.451,148.742
C03131=1100.885,-109.092,-47.475,179.969,4.446,148.741
C03132=1100.890,-109.342,-47.464,179.969,4.441,148.740
C03133=1100.895,-109.592,-47.454,179.970,4.436,148.739
C03134=1100.901,-109.842,-47.444,179.970,4.431,148.737
C03135=1100.906,-110.092,-47.433,179.971,4.426,148.736
C03136=1100.911,-110.341,-47.423,179.971,4.420,148.735
C03137=1100.916,-110.591,-47.413,179.972,4.416,148.734
C03138=1100.921,-110.841,-47.403,179.972,4.411,148.732
C03139=1100.927,-111.090,-47.393,179.973,4.406,148.731
C03140=1100.933,-111.340,-47.382,179.974,4.401,148.730
C03141=1100.938,-111.590,-47.372,179.974,4.396,148.728
C03142=1100.943,-111.840,-47.362,179.974,4.391,148.727
C03143=1100.948,-112.089,-47.352,179.975,4.386,148.726
C03144=1100.953,-112.339,-47.341,179.976,4.381,148.725
C03145=1100.959,-112.589,-47.331,179.976,4.376,148.723
C03146=1100.964,-112.839,-47.321,179.977,4.371,148.722
C03147=1100.968,-113.053,-47.312,179.977,4.366,148.721
C03148=1100.972,-113.267,-47.303,179.978,4.362,148.720
C03149=1100.977,-113.482,-47.295,179.978,4.357,148.719
C03150=1100.981,-113.696,-47.286,179.978,4.353,148.718
C03151=1100.986,-113.910,-47.277,179.979,4.349,148.717
C03152=1100.991,-114.125,-47.269,179.980,4.345,148.716
C03153=1100.995,-114.339,-47.260,179.980,4.340,148.714
C03154=1100.999,-114.553,-47.251,179.980,4.336,148.713
C03155=1101.005,-114.803,-47.241,179.981,4.330,148.712
C03156=1101.010,-115.053,-47.230,179.982,4.326,148.711
C03157=1101.015,-115.302,-47.221,179.982,4.321,148.710
C03158=1101.021,-115.552,-47.211,179.982,4.316,148.708
C03159=1101.026,-115.803,-47.201,179.983,4.310,148.707
C03160=1101.031,-116.052,-47.191,179.984,4.306,148.706
C03161=1101.036,-116.301,-47.181,179.984,4.301,148.704
C03162=1101.042,-116.551,-47.171,179.985,4.295,148.703
C03163=1101.047,-116.801,-47.160,179.985,4.290,148.702
C03164=1101.052,-117.050,-47.150,179.985,4.285,148.701
C03165=1101.058,-117.301,-47.141,179.987,4.280,148.699
C03166=1101.063,-117.551,-47.130,179.987,4.275,148.698
C03167=1101.067,-117.800,-47.121,179.987,4.270,148.697
C03168=1101.073,-118.050,-47.111,179.988,4.264,148.695
C03169=1101.079,-118.299,-47.100,179.988,4.259,148.694
C03170=1101.083,-118.550,-47.091,179.990,4.254,148.692
C03171=1101.089,-118.799,-47.081,179.990,4.249,148.691
C03172=1101.094,-119.049,-47.071,179.990,4.244,148.690
C03173=1101.099,-119.298,-47.061,179.991,4.239,148.689
C03174=1101.104,-119.548,-47.051,179.991,4.233,148.687
C03175=1101.110,-119.798,-47.041,179.992,4.229,148.686
C03176=1101.115,-120.048,-47.031,179.993,4.224,148.685
C03177=1101.121,-120.297,-47.021,179.993,4.218,148.683
C03178=1101.125,-120.547,-47.011,179.994,4.213,148.682
C03179=1101.131,-120.797,-47.002,179.994,4.208,148.681
C03180=1101.136,-121.047,-46.992,179.995,4.202,148.679
C03181=1101.141,-121.296,-46.982,179.996,4.198,148.678
C03182=1101.147,-121.546,-46.972,179.996,4.193,148.677
C03183=1101.151,-121.796,-46.962,179.997,4.187,148.675
C03184=1101.157,-122.046,-46.952,179.998,4.182,148.674
C03185=1101.163,-122.295,-46.942,179.998,4.176,148.673
C03186=1101.168,-122.545,-46.933,179.999,4.171,148.672
C03187=1101.173,-122.795,-46.923,179.999,4.166,148.670
C03188=1101.178,-123.045,-46.913,-180.000,4.161,148.669
C03189=1101.184,-123.295,-46.903,-179.999,4.156,148.667
C03190=1101.188,-123.544,-46.894,-179.999,4.151,148.666
C03191=1101.194,-123.793,-46.884,-179.998,4.145,148.665
C03192=1101.199,-124.043,-46.875,-179.998,4.140,148.663
C03193=1101.204,-124.294,-46.864,-179.997,4.135,148.662
C03194=1101.210,-124.544,-46.855,-179.996,4.129,148.661
C03195=1101.215,-124.793,-46.845,-179.995,4.125,148.659
C03196=1101.221,-125.042,-46.835,-179.995,4.120,148.658
C03197=1101.226,-125.292,-46.826,-179.994,4.114,148.657
C03198=1101.231,-125.542,-46.816,-179.993,4.108,148.655
C03199=1101.236,-125.792,-46.806,-179.993,4.103,148.654
C03200=1101.242,-126.042,-46.796,-179.992,4.098,148.652
C03201=1101.246,-126.291,-46.787,-179.992,4.093,148.651
C03202=1101.252,-126.541,-46.777,-179.991,4.087,148.650
C03203=1101.257,-126.756,-46.769,-179.990,4.083,148.648
C03204=1101.261,-126.970,-46.760,-179.989,4.078,148.647
C03205=1101.266,-127.185,-46.752,-179.989,4.074,148.646
C03206=1101.270,-127.399,-46.744,-179.988,4.069,148.645
C03207=1101.274,-127.613,-46.736,-179.988,4.065,148.644
C03208=1101.279,-127.828,-46.728,-179.987,4.060,148.643
C03209=1101.283,-128.042,-46.719,-179.986,4.055,148.641
C03210=1101.288,-128.257,-46.711,-179.986,4.050,148.640
C03211=1100.865,-128.248,-46.737,-179.979,4.055,148.639
C03212=1100.860,-128.033,-46.746,-179.979,4.060,148.640
C03213=1100.856,-127.819,-46.754,-179.980,4.064,148.641
C03214=1100.851,-127.604,-46.762,-179.981,4.069,148.643
C03215=1100.847,-127.390,-46.771,-179.981,4.074,148.644
C03216=1100.842,-127.175,-46.779,-179.982,4.078,148.645
C03217=1100.838,-126.961,-46.787,-179.982,4.082,148.646
C03218=1100.833,-126.746,-46.796,-179.983,4.087,148.647
C03219=1100.829,-126.532,-46.804,-179.984,4.092,148.648
C03220=1100.824,-126.282,-46.813,-179.984,4.097,148.650
C03221=1100.818,-126.032,-46.823,-179.985,4.102,148.651
C03222=1100.813,-125.783,-46.832,-179.985,4.108,148.652
C03223=1100.807,-125.533,-46.842,-179.986,4.113,148.654
C03224=1100.803,-125.283,-46.852,-179.987,4.118,148.655
C03225=1100.797,-125.033,-46.862,-179.988,4.123,148.657
C03226=1100.792,-124.784,-46.871,-179.988,4.129,148.658
C03227=1100.787,-124.534,-46.882,-179.989,4.134,148.659
C03228=1100.782,-124.284,-46.890,-179.990,4.139,148.661
C03229=1100.777,-124.034,-46.901,-179.990,4.144,148.662
C03230=1100.771,-123.784,-46.910,-179.991,4.150,148.663
C03231=1100.766,-123.535,-46.920,-179.991,4.154,148.665
C03232=1100.760,-123.285,-46.930,-179.992,4.160,148.666
C03233=1100.755,-123.036,-46.940,-179.993,4.165,148.667
C03234=1100.750,-122.785,-46.950,-179.993,4.170,148.669
C03235=1100.745,-122.536,-46.959,-179.994,4.176,148.670
C03236=1100.740,-122.286,-46.970,-179.994,4.181,148.672
C03237=1100.734,-122.036,-46.979,-179.995,4.186,148.673
C03238=1100.729,-121.787,-46.989,-179.996,4.191,148.674
C03239=1100.724,-121.537,-46.999,-179.996,4.196,148.675
C03240=1100.719,-121.287,-47.009,-179.997,4.202,148.677
C03241=1100.713,-121.037,-47.018,-179.998,4.207,148.678
C03242=1100.707,-120.788,-47.029,-179.998,4.212,148.680
C03243=1100.703,-120.538,-47.039,-179.999,4.217,148.681
C03244=1100.698,-120.288,-47.049,-179.999,4.222,148.682
C03245=1100.692,-120.038,-47.058,180.000,4.227,148.683
C03246=1100.687,-119.789,-47.068,179.999,4.233,148.685
C03247=1100.682,-119.539,-47.079,179.999,4.238,148.686
C03248=1100.677,-119.289,-47.088,179.998,4.243,148.687
C03249=1100.671,-119.039,-47.098,179.998,4.248,148.689
C03250=1100.665,-118.790,-47.108,179.997,4.253,148.690
C03251=1100.661,-118.540,-47.118,179.996,4.258,148.691
C03252=1100.656,-118.290,-47.128,179.996,4.264,148.693
C03253=1100.650,-118.041,-47.138,179.995,4.269,148.694
C03254=1100.646,-117.791,-47.148,179.995,4.273,148.695
C03255=1100.640,-117.540,-47.158,179.994,4.279,148.697
C03256=1100.634,-117.291,-47.168,179.993,4.284,148.698
C03257=1100.629,-117.041,-47.178,179.993,4.289,148.699
C03258=1100.624,-116.791,-47.188,179.992,4.294,148.701
C03259=1100.619,-116.542,-47.198,179.992,4.299,148.702
C03260=1100.613,-116.292,-47.209,179.991,4.304,148.703
C03261=1100.609,-116.042,-47.218,179.991,4.310,148.704
C03262=1100.603,-115.793,-47.229,179.990,4.315,148.706
C03263=1100.597,-115.543,-47.238,179.989,4.319,148.707
C03264=1100.592,-115.293,-47.248,179.989,4.325,148.708
C03265=1100.588,-115.043,-47.258,179.988,4.330,148.710
C03266=1100.582,-114.794,-47.269,179.988,4.335,148.711
C03267=1100.576,-114.544,-47.279,179.987,4.340,148.712
C03268=1100.572,-114.330,-47.287,179.987,4.344,148.713
C03269=1100.568,-114.115,-47.297,179.986,4.349,148.714
C03270=1100.564,-113.901,-47.305,179.986,4.353,148.715
C03271=1100.559,-113.686,-47.314,179.985,4.357,148.717
C03272=1100.554,-113.472,-47.323,179.985,4.362,148.718
C03273=1100.550,-113.258,-47.331,179.984,4.366,148.719
C03274=1100.546,-113.044,-47.340,179.984,4.370,148.720
C03275=1100.541,-112.829,-47.349,179.983,4.374,148.721
C03276=1100.536,-112.580,-47.359,179.983,4.380,148.722
C03277=1100.531,-112.330,-47.369,179.983,4.385,148.723
C03278=1100.525,-112.080,-47.380,179.981,4.389,148.725
C03279=1100.519,-111.830,-47.390,179.981,4.395,148.726
C03280=1100.515,-111.581,-47.400,179.981,4.400,148.727
C03281=1100.509,-111.331,-47.410,179.981,4.405,148.728
C03282=1100.504,-111.081,-47.420,179.980,4.409,148.730
C03283=1100.499,-110.831,-47.431,179.979,4.415,148.731
C03284=1100.493,-110.582,-47.441,179.979,4.420,148.732
C03285=1100.488,-110.331,-47.451,179.978,4.425,148.734
C03286=1100.483,-110.082,-47.461,179.978,4.429,148.735
C03287=1100.478,-109.833,-47.471,179.977,4.434,148.736
C03288=1100.473,-109.582,-47.482,179.977,4.440,148.737
C03289=1100.467,-109.333,-47.492,179.976,4.445,148.739
C03290=1100.463,-109.083,-47.503,179.976,4.449,148.740
C03291=1100.457,-108.834,-47.514,179.975,4.455,148.741
C03292=1100.451,-108.584,-47.524,179.975,4.460,148.742
C03293=1100.446,-108.334,-47.534,179.974,4.464,148.744
C03294=1100.441,-108.085,-47.544,179.973,4.470,148.745
C03295=1100.436,-107.834,-47.555,179.973,4.475,148.746
C03296=1100.431,-107.585,-47.565,179.973,4.480,148.747
C03297=1100.426,-107.335,-47.575,179.972,4.484,148.748
C03298=1100.420,-107.085,-47.586,179.972,4.489,148.750
C03299=1100.415,-106.836,-47.596,179.971,4.495,148.751
C03300=1100.410,-106.586,-47.607,179.970,4.499,148.752
C03301=1100.404,-106.336,-47.617,179.970,4.504,148.754
C03302=1100.399,-106.086,-47.628,179.970,4.510,148.755
C03303=1100.394,-105.837,-47.638,179.969,4.514,148.756
C03304=1100.390,-105.587,-47.649,179.969,4.519,148.757
C03305=1100.384,-105.338,-47.659,179.969,4.524,148.758
C03306=1100.379,-105.087,-47.670,179.968,4.529,148.760
C03307=1100.374,-104.838,-47.680,179.967,4.534,148.761
C03308=1100.369,-104.588,-47.690,179.967,4.539,148.762
C03309=1100.363,-104.339,-47.701,179.967,4.544,148.763
C03310=1100.358,-104.089,-47.711,179.966,4.549,148.765
C03311=1100.353,-103.839,-47.722,179.966,4.554,148.766
C03312=1100.347,-103.589,-47.732,179.965,4.559,148.767
C03313=1100.342,-103.340,-47.744,179.964,4.563,148.768
C03314=1100.337,-103.090,-47.754,179.964,4.568,148.769
C03315=1100.332,-102.840,-47.764,179.964,4.574,148.771
C03316=1100.326,-102.590,-47.775,179.963,4.578,148.772
C03317=1100.322,-102.341,-47.786,179.962,4.583,148.773
C03318=1100.316,-102.091,-47.796,179.962,4.589,148.775
C03319=1100.311,-101.841,-47.807,179.962,4.594,148.776
C03320=1100.305,-101.592,-47.817,179.961,4.598,148.777
C03321=1100.301,-101.342,-47.828,179.961,4.603,148.778
C03322=1100.295,-101.092,-47.838,179.961,4.608,148.779
C03323=1100.290,-100.842,-47.849,179.960,4.613,148.781
C03324=1100.285,-100.628,-47.859,179.960,4.617,148.781
C03325=1100.281,-100.414,-47.868,179.959,4.622,148.783
C03326=1100.277,-100.200,-47.877,179.959,4.626,148.784
C03327=1100.272,-99.985,-47.886,179.959,4.630,148.785
C03328=1100.268,-99.771,-47.895,179.958,4.634,148.786
C03329=1100.263,-99.557,-47.905,179.958,4.638,148.787
C03330=1100.259,-99.343,-47.914,179.957,4.642,148.788
C03331=1100.254,-99.128,-47.923,179.957,4.646,148.789
C03332=1100.249,-98.879,-47.934,179.956,4.651,148.790
C03333=1100.244,-98.628,-47.944,179.956,4.657,148.791
C03334=1100.238,-98.379,-47.955,179.956,4.662,148.793
C03335=1100.234,-98.129,-47.966,179.955,4.666,148.794
C03336=1100.228,-97.880,-47.976,179.955,4.671,148.795
C03337=1100.223,-97.630,-47.987,179.955,4.676,148.796
C03338=1100.218,-97.380,-47.998,179.954,4.681,148.797
C03339=1100.213,-97.131,-48.009,179.954,4.686,148.798
C03340=1100.207,-96.881,-48.019,179.954,4.691,148.800
C03341=1100.202,-96.631,-48.030,179.953,4.695,148.801
C03342=1100.197,-96.381,-48.042,179.953,4.700,148.802
C03343=1100.191,-96.132,-48.052,179.952,4.706,148.803
C03344=1100.187,-95.882,-48.063,179.952,4.710,148.804
C03345=1100.181,-95.632,-48.073,179.951,4.715,148.806
C03346=1100.176,-95.383,-48.085,179.951,4.720,148.807
C03347=1100.171,-95.132,-48.095,179.950,4.724,148.808
C03348=1100.165,-94.883,-48.107,179.950,4.730,148.809
C03349=1100.160,-94.633,-48.117,179.949,4.735,148.811
C03350=1100.155,-94.384,-48.128,179.949,4.739,148.812
C03351=1100.150,-94.134,-48.139,179.948,4.745,148.813
C03352=1100.145,-93.884,-48.150,179.948,4.750,148.814
C03353=1100.139,-93.634,-48.161,179.948,4.754,148.815
C03354=1100.134,-93.385,-48.172,179.948,4.759,148.816
C03355=1100.129,-93.135,-48.182,179.948,4.764,148.818
C03356=1100.124,-92.886,-48.194,179.947,4.769,148.819
C03357=1100.119,-92.636,-48.205,179.947,4.773,148.820
C03358=1100.113,-92.386,-48.216,179.946,4.779,148.821
C03359=1100.108,-92.136,-48.227,179.946,4.784,148.822
C03360=1100.103,-91.886,-48.238,179.946,4.789,148.824
C03361=1100.098,-91.637,-48.248,179.946,4.794,148.825
C03362=1100.093,-91.387,-48.259,179.945,4.798,148.826
C03363=1100.088,-91.137,-48.271,179.945,4.803,148.827
C03364=1100.082,-90.888,-48.282,179.945,4.809,148.828
C03365=1100.077,-90.638,-48.292,179.944,4.814,148.830
C03366=1100.073,-90.388,-48.304,179.944,4.819,148.831
C03367=1100.067,-90.139,-48.315,179.944,4.824,148.832
C03368=1100.062,-89.889,-48.326,179.943,4.828,148.833
C03369=1100.057,-89.639,-48.337,179.943,4.834,148.835
C03370=1100.052,-89.390,-48.348,179.942,4.839,148.836
C03371=1100.046,-89.140,-48.359,179.942,4.844,148.837
C03372=1100.041,-88.890,-48.371,179.942,4.849,148.838
C03373=1100.036,-88.641,-48.381,179.942,4.854,148.839
C03374=1100.030,-88.391,-48.393,179.941,4.859,148.840
C03375=1100.025,-88.141,-48.404,179.941,4.864,148.842
C03376=1100.021,-87.891,-48.415,179.941,4.869,148.843
C03377=1100.014,-87.641,-48.426,179.940,4.874,148.844
C03378=1100.010,-87.392,-48.437,179.940,4.879,148.845
C03379=1100.005,-87.142,-48.449,179.940,4.884,148.846
C03380=1100.000,-86.928,-48.458,179.940,4.888,148.847
C03381=1099.996,-86.714,-48.467,179.939,4.893,148.849
C03382=1099.992,-86.499,-48.477,179.939,4.897,148.849
C03383=1099.987,-86.285,-48.487,179.939,4.902,148.851
C03384=1099.982,-86.071,-48.496,179.938,4.906,148.852
C03385=1099.978,-85.857,-48.507,179.939,4.911,148.853
C03386=1099.973,-85.643,-48.516,179.938,4.915,148.854
C03387=1099.969,-85.429,-48.525,179.938,4.919,148.855
C03388=1099.964,-85.179,-48.537,179.937,4.924,148.856
C03389=1099.959,-84.929,-48.548,179.937,4.929,148.857
C03390=1099.954,-84.679,-48.559,179.937,4.934,148.858
C03391=1099.948,-84.430,-48.571,179.937,4.939,148.859
C03392=1099.943,-84.181,-48.582,179.936,4.945,148.861
C03393=1099.938,-83.931,-48.594,179.936,4.950,148.862
C03394=1099.933,-83.681,-48.605,179.936,4.955,148.863
C03395=1099.928,-83.431,-48.615,179.936,4.960,148.864
C03396=1099.922,-83.181,-48.627,179.935,4.965,148.866
C03397=1099.918,-82.932,-48.638,179.935,4.970,148.867
C03398=1099.912,-82.682,-48.650,179.935,4.975,148.868
C03399=1099.907,-82.433,-48.661,179.935,4.980,148.869
C03400=1099.901,-82.183,-48.673,179.934,4.985,148.870
C03401=1099.897,-81.933,-48.684,179.934,4.990,148.872
C03402=1099.891,-81.683,-48.696,179.933,4.996,148.873
C03403=1099.887,-81.434,-48.708,179.933,5.001,148.874
C03404=1099.881,-81.184,-48.718,179.933,5.006,148.875
C03405=1099.876,-80.934,-48.730,179.933,5.011,148.876
C03406=1099.871,-80.685,-48.741,179.933,5.016,148.878
C03407=1099.865,-80.435,-48.753,179.933,5.021,148.879
C03408=1099.861,-80.185,-48.764,179.932,5.026,148.880
C03409=1099.855,-79.935,-48.776,179.932,5.031,148.881
C03410=1099.850,-79.686,-48.787,179.932,5.036,148.882
C03411=1099.845,-79.436,-48.799,179.931,5.041,148.884
C03412=1099.840,-79.187,-48.810,179.931,5.047,148.885
C03413=1099.835,-78.937,-48.822,179.931,5.052,148.886
C03414=1099.830,-78.687,-48.833,179.930,5.057,148.887
C03415=1099.824,-78.437,-48.845,179.930,5.062,148.889
C03416=1099.818,-78.188,-48.857,179.930,5.067,148.890
C03417=1099.814,-77.938,-48.868,179.930,5.072,148.891
C03418=1099.808,-77.688,-48.880,179.930,5.078,148.892
C03419=1099.804,-77.439,-48.891,179.930,5.083,148.893
C03420=1099.798,-77.189,-48.903,179.930,5.088,148.894
C03421=1099.793,-76.939,-48.914,179.929,5.092,148.896
C03422=1099.788,-76.689,-48.926,179.929,5.097,148.897
C03423=1099.782,-76.440,-48.938,179.928,5.102,148.898
C03424=1099.777,-76.190,-48.949,179.928,5.108,148.899
C03425=1099.772,-75.941,-48.962,179.928,5.113,148.901
C03426=1099.767,-75.692,-48.973,179.928,5.118,148.902
C03427=1099.762,-75.442,-48.985,179.927,5.123,148.903
C03428=1099.757,-75.192,-48.997,179.927,5.128,148.904
C03429=1099.752,-74.942,-49.008,179.927,5.134,148.905
C03430=1099.746,-74.692,-49.020,179.927,5.139,148.906
C03431=1099.742,-74.442,-49.031,179.927,5.144,148.908
C03432=1099.736,-74.193,-49.043,179.927,5.149,148.909
C03433=1099.731,-73.944,-49.055,179.927,5.154,148.910
C03434=1099.726,-73.694,-49.067,179.926,5.159,148.911
C03435=1099.721,-73.444,-49.078,179.926,5.164,148.912
C03436=1099.714,-73.128,-49.094,179.926,5.171,148.914
C03437=1099.708,-72.811,-49.108,179.926,5.176,148.915
C03438=1099.700,-72.495,-49.123,179.925,5.183,148.917
C03439=1099.695,-72.179,-49.138,179.925,5.189,148.918
C03440=1099.689,-71.929,-49.150,179.925,5.194,148.919
C03441=1099.684,-71.679,-49.162,179.925,5.199,148.921
C03442=1099.679,-71.429,-49.174,179.925,5.205,148.922
C03443=1099.674,-71.180,-49.186,179.924,5.210,148.923
C03444=1099.669,-70.930,-49.198,179.924,5.215,148.924
C03445=1099.663,-70.681,-49.210,179.924,5.220,148.925
C03446=1099.659,-70.431,-49.221,179.924,5.225,148.926
C03447=1099.653,-70.182,-49.234,179.924,5.230,148.928
C03448=1099.648,-69.932,-49.245,179.924,5.235,148.929
C03449=1099.643,-69.682,-49.257,179.924,5.241,148.930
C03450=1099.638,-69.433,-49.269,179.924,5.245,148.931
C03451=1099.633,-69.183,-49.281,179.923,5.250,148.932
C03452=1099.627,-68.933,-49.293,179.923,5.255,148.933
C03453=1099.622,-68.683,-49.306,179.923,5.260,148.934
C03454=1099.618,-68.434,-49.317,179.923,5.265,148.936
C03455=1099.612,-68.184,-49.329,179.923,5.270,148.937
C03456=1099.607,-67.935,-49.342,179.923,5.275,148.938
C03457=1099.602,-67.685,-49.353,179.922,5.280,148.939
C03458=1099.597,-67.435,-49.365,179.923,5.285,148.940
C03459=1099.592,-67.186,-49.377,179.923,5.290,148.941
C03460=1099.586,-66.936,-49.389,179.923,5.295,148.942
C03461=1099.581,-66.686,-49.401,179.922,5.300,148.943
C03462=1099.576,-66.437,-49.414,179.922,5.305,148.945
C03463=1099.571,-66.187,-49.425,179.922,5.310,148.946
C03464=1099.566,-65.938,-49.438,179.922,5.315,148.947
C03465=1099.561,-65.688,-49.449,179.922,5.320,148.948
C03466=1099.555,-65.438,-49.462,179.922,5.325,148.949
C03467=1099.550,-65.188,-49.474,179.922,5.330,148.950
C03468=1099.545,-64.938,-49.486,179.922,5.335,148.951
C03469=1099.540,-64.689,-49.498,179.922,5.340,148.952
C03470=1099.535,-64.440,-49.510,179.921,5.344,148.953
C03471=1099.530,-64.190,-49.523,179.922,5.349,148.954
C03472=1099.525,-63.940,-49.535,179.922,5.354,148.956
C03473=1099.520,-63.690,-49.547,179.921,5.359,148.957
C03474=1099.514,-63.440,-49.559,179.922,5.364,148.958
C03475=1099.509,-63.191,-49.572,179.922,5.369,148.959
C03476=1099.283,-72.673,-49.148,179.932,5.184,148.915
C03477=1099.290,-73.054,-49.130,179.932,5.176,148.913
C03478=1099.299,-73.435,-49.113,179.933,5.168,148.911
C03479=1099.304,-73.685,-49.100,179.933,5.163,148.910
C03480=1099.309,-73.935,-49.088,179.933,5.158,148.909
C03481=1099.314,-74.184,-49.077,179.933,5.153,148.908
C03482=1099.319,-74.434,-49.065,179.933,5.148,148.906
C03483=1099.325,-74.684,-49.053,179.934,5.142,148.905
C03484=1099.329,-74.933,-49.041,179.934,5.137,148.904
C03485=1099.334,-75.183,-49.029,179.934,5.132,148.903
C03486=1099.339,-75.433,-49.018,179.934,5.127,148.902
C03487=1099.345,-75.683,-49.006,179.934,5.122,148.901
C03488=1099.350,-75.933,-48.994,179.934,5.117,148.899
C03489=1099.355,-76.182,-48.983,179.934,5.112,148.898
C03490=1099.361,-76.432,-48.971,179.935,5.106,148.897
C03491=1099.366,-76.681,-48.959,179.936,5.102,148.896
C03492=1099.371,-76.931,-48.948,179.936,5.097,148.894
C03493=1099.376,-77.180,-48.935,179.936,5.092,148.893
C03494=1099.381,-77.430,-48.924,179.936,5.086,148.892
C03495=1099.386,-77.680,-48.912,179.936,5.081,148.891
C03496=1099.391,-77.930,-48.901,179.937,5.076,148.890
C03497=1099.396,-78.180,-48.889,179.937,5.071,148.889
C03498=1099.402,-78.429,-48.878,179.937,5.066,148.887
C03499=1099.407,-78.678,-48.866,179.937,5.061,148.886
C03500=1099.412,-78.928,-48.854,179.937,5.056,148.885
C03501=1099.417,-79.178,-48.843,179.937,5.050,148.884
C03502=1099.422,-79.428,-48.831,179.938,5.045,148.883
C03503=1099.427,-79.678,-48.820,179.938,5.040,148.881
C03504=1099.433,-79.927,-48.808,179.938,5.035,148.880
C03505=1099.438,-80.176,-48.797,179.939,5.030,148.879
C03506=1099.443,-80.426,-48.785,179.939,5.025,148.878
C03507=1099.448,-80.676,-48.774,179.939,5.020,148.876
C03508=1099.453,-80.926,-48.762,179.940,5.015,148.875
C03509=1099.458,-81.176,-48.751,179.940,5.010,148.874
C03510=1099.464,-81.425,-48.739,179.940,5.005,148.873
C03511=1099.469,-81.674,-48.728,179.940,5.000,148.872
C03512=1099.474,-81.924,-48.716,179.941,4.994,148.870
C03513=1099.479,-82.174,-48.705,179.941,4.989,148.869
C03514=1099.485,-82.425,-48.694,179.941,4.984,148.868
C03515=1099.489,-82.674,-48.682,179.941,4.979,148.867
C03516=1099.495,-82.923,-48.671,179.941,4.974,148.866
C03517=1099.500,-83.173,-48.660,179.942,4.969,148.864
C03518=1099.506,-83.423,-48.648,179.942,4.964,148.863
C03519=1099.510,-83.673,-48.636,179.943,4.959,148.862
C03520=1099.516,-83.921,-48.625,179.943,4.954,148.861
C03521=1099.521,-84.171,-48.614,179.943,4.949,148.860
C03522=1099.526,-84.422,-48.603,179.944,4.943,148.858
C03523=1099.531,-84.672,-48.591,179.944,4.938,148.857
C03524=1099.536,-84.921,-48.580,179.944,4.933,148.856
C03525=1099.541,-85.170,-48.569,179.944,4.928,148.855
C03526=1099.547,-85.420,-48.557,179.945,4.923,148.854
C03527=1099.551,-85.634,-48.548,179.945,4.919,148.853
C03528=1099.555,-85.849,-48.538,179.945,4.914,148.851
C03529=1099.560,-86.063,-48.528,179.946,4.910,148.850
C03530=1099.564,-86.277,-48.519,179.945,4.906,148.849
C03531=1099.569,-86.491,-48.509,179.946,4.901,148.848
C03532=1099.573,-86.705,-48.499,179.946,4.897,148.847
C03533=1099.578,-86.919,-48.490,179.946,4.893,148.846
C03534=1099.582,-87.134,-48.480,179.947,4.888,148.845
C03535=1099.587,-87.383,-48.469,179.947,4.883,148.844
C03536=1099.593,-87.633,-48.457,179.947,4.878,148.843
C03537=1099.598,-87.883,-48.447,179.947,4.873,148.842
C03538=1099.602,-88.133,-48.435,179.947,4.868,148.840
C03539=1099.608,-88.382,-48.424,179.948,4.863,148.839
C03540=1099.613,-88.631,-48.412,179.948,4.858,148.838
C03541=1099.618,-88.882,-48.402,179.949,4.853,148.837
C03542=1099.624,-89.131,-48.390,179.949,4.848,148.836
C03543=1099.629,-89.381,-48.379,179.949,4.843,148.835
C03544=1099.634,-89.631,-48.368,179.949,4.838,148.833
C03545=1099.639,-89.880,-48.358,179.949,4.833,148.832
C03546=1099.645,-90.130,-48.346,179.950,4.828,148.831
C03547=1099.650,-90.380,-48.335,179.951,4.823,148.830
C03548=1099.654,-90.630,-48.324,179.951,4.818,148.828
C03549=1099.660,-90.879,-48.312,179.951,4.812,148.827
C03550=1099.665,-91.129,-48.302,179.951,4.807,148.826
C03551=1099.670,-91.379,-48.290,179.952,4.802,148.825
C03552=1099.675,-91.628,-48.279,179.952,4.798,148.824
C03553=1099.681,-91.878,-48.268,179.953,4.793,148.822
C03554=1099.686,-92.128,-48.257,179.953,4.788,148.821
C03555=1099.691,-92.377,-48.247,179.953,4.782,148.820
C03556=1099.696,-92.627,-48.236,179.953,4.777,148.819
C03557=1099.701,-92.877,-48.224,179.953,4.773,148.818
C03558=1099.707,-93.126,-48.213,179.954,4.768,148.817
C03559=1099.712,-93.376,-48.202,179.954,4.763,148.815
C03560=1099.717,-93.626,-48.192,179.954,4.758,148.814
C03561=1099.722,-93.875,-48.181,179.954,4.753,148.813
C03562=1099.727,-94.125,-48.170,179.955,4.748,148.812
C03563=1099.733,-94.375,-48.159,179.955,4.743,148.811
C03564=1099.738,-94.625,-48.148,179.955,4.738,148.809
C03565=1099.743,-94.875,-48.137,179.956,4.734,148.808
C03566=1099.748,-95.123,-48.126,179.956,4.729,148.807
C03567=1099.753,-95.374,-48.115,179.957,4.724,148.806
C03568=1099.759,-95.623,-48.104,179.957,4.719,148.805
C03569=1099.764,-95.873,-48.093,179.958,4.714,148.804
C03570=1099.769,-96.123,-48.082,179.958,4.709,148.802
C03571=1099.774,-96.372,-48.072,179.959,4.704,148.801
C03572=1099.779,-96.623,-48.061,179.959,4.699,148.800
C03573=1099.785,-96.872,-48.050,179.960,4.694,148.798
C03574=1099.790,-97.122,-48.040,179.960,4.690,148.797
C03575=1099.795,-97.372,-48.028,179.961,4.684,148.796
C03576=1099.801,-97.621,-48.017,179.961,4.679,148.795
C03577=1099.805,-97.871,-48.006,179.962,4.675,148.794
C03578=1099.811,-98.120,-47.996,179.962,4.670,148.792
C03579=1099.816,-98.370,-47.985,179.962,4.665,148.791
C03580=1099.821,-98.620,-47.974,179.963,4.660,148.790
C03581=1099.826,-98.870,-47.964,179.963,4.655,148.789
C03582=1099.831,-99.119,-47.953,179.963,4.650,148.788
C03583=1099.836,-99.334,-47.943,179.964,4.646,148.787
C03584=1099.840,-99.548,-47.935,179.964,4.642,148.786
C03585=1099.845,-99.762,-47.925,179.965,4.638,148.785
C03586=1099.849,-99.976,-47.916,179.965,4.634,148.784
C03587=1099.854,-100.190,-47.906,179.966,4.630,148.782
C03588=1099.858,-100.405,-47.897,179.966,4.626,148.781
C03589=1099.863,-100.619,-47.889,179.966,4.621,148.781
C03590=1099.867,-100.833,-47.879,179.967,4.616,148.779
C03591=1099.873,-101.083,-47.869,179.967,4.612,148.778
C03592=1099.878,-101.333,-47.857,179.968,4.607,148.777
C03593=1099.883,-101.582,-47.847,179.968,4.602,148.776
C03594=1099.888,-101.832,-47.837,179.969,4.598,148.775
C03595=1099.893,-102.082,-47.825,179.969,4.592,148.773
C03596=1099.899,-102.332,-47.815,179.969,4.587,148.772
C03597=1099.904,-102.582,-47.805,179.969,4.582,148.771
C03598=1099.909,-102.831,-47.794,179.970,4.578,148.770
C03599=1099.914,-103.081,-47.783,179.971,4.572,148.768
C03600=1099.920,-103.330,-47.773,179.971,4.567,148.767
C03601=1099.925,-103.581,-47.762,179.972,4.563,148.766
C03602=1099.930,-103.830,-47.751,179.972,4.558,148.765
C03603=1099.935,-104.080,-47.741,179.972,4.552,148.763
C03604=1099.940,-104.329,-47.731,179.973,4.548,148.762
C03605=1099.945,-104.579,-47.719,179.973,4.543,148.761
C03606=1099.951,-104.829,-47.709,179.974,4.538,148.760
C03607=1099.956,-105.079,-47.698,179.974,4.534,148.759
C03608=1099.961,-105.328,-47.688,179.975,4.528,148.757
C03609=1099.967,-105.578,-47.678,179.975,4.523,148.756
C03610=1099.972,-105.828,-47.667,179.976,4.519,148.755
C03611=1099.977,-106.077,-47.657,179.976,4.513,148.754
C03612=1099.982,-106.327,-47.646,179.977,4.508,148.752
C03613=1099.988,-106.577,-47.636,179.977,4.503,148.751
C03614=1099.993,-106.827,-47.625,179.978,4.499,148.750
C03615=1099.998,-107.076,-47.614,179.979,4.493,148.748
C03616=1100.002,-107.326,-47.604,179.979,4.488,148.747
C03617=1100.008,-107.576,-47.594,179.980,4.484,148.746
C03618=1100.013,-107.826,-47.584,179.980,4.479,148.745
C03619=1100.019,-108.075,-47.573,179.980,4.473,148.744
C03620=1100.024,-108.325,-47.563,179.981,4.469,148.742
C03621=1100.029,-108.574,-47.552,179.982,4.464,148.741
C03622=1100.034,-108.824,-47.542,179.982,4.458,148.740
C03623=1100.039,-109.074,-47.531,179.982,4.453,148.739
C03624=1100.045,-109.324,-47.521,179.983,4.449,148.737
C03625=1100.049,-109.574,-47.511,179.983,4.444,148.736
C03626=1100.055,-109.823,-47.501,179.984,4.438,148.735
C03627=1100.060,-110.073,-47.490,179.984,4.433,148.734
C03628=1100.065,-110.323,-47.480,179.985,4.429,148.732
C03629=1100.071,-110.573,-47.470,179.985,4.424,148.731
C03630=1100.076,-110.823,-47.459,179.986,4.419,148.730
C03631=1100.082,-111.072,-47.449,179.987,4.414,148.728
C03632=1100.086,-111.321,-47.439,179.987,4.409,148.727
C03633=1100.091,-111.571,-47.428,179.987,4.404,148.726
C03634=1100.097,-111.821,-47.418,179.988,4.398,148.725
C03635=1100.102,-112.071,-47.407,179.989,4.394,148.723
C03636=1100.107,-112.321,-47.397,179.989,4.389,148.722
C03637=1100.113,-112.570,-47.387,179.990,4.383,148.721
C03638=1100.117,-112.820,-47.377,179.990,4.378,148.720
C03639=1100.123,-113.035,-47.368,179.991,4.374,148.718
C03640=1100.127,-113.249,-47.359,179.991,4.370,148.718
C03641=1100.131,-113.463,-47.350,179.992,4.366,148.716
C03642=1100.136,-113.678,-47.342,179.992,4.362,148.715
C03643=1100.140,-113.891,-47.333,179.992,4.356,148.714
C03644=1100.145,-114.106,-47.324,179.993,4.353,148.713
C03645=1100.149,-114.320,-47.315,179.994,4.348,148.712
C03646=1100.154,-114.535,-47.307,179.994,4.344,148.711
C03647=1100.159,-114.784,-47.297,179.995,4.339,148.710
C03648=1100.164,-115.034,-47.286,179.995,4.334,148.708
C03649=1100.169,-115.284,-47.276,179.995,4.328,148.707
C03650=1100.175,-115.533,-47.266,179.997,4.324,148.706
C03651=1100.180,-115.783,-47.256,179.997,4.319,148.704
C03652=1100.186,-116.033,-47.245,179.997,4.313,148.703
C03653=1100.191,-116.283,-47.237,179.998,4.308,148.702
C03654=1100.196,-116.533,-47.226,179.999,4.304,148.701
C03655=1100.201,-116.783,-47.216,179.999,4.298,148.699
C03656=1100.207,-117.032,-47.206,180.000,4.293,148.698
C03657=1100.211,-117.282,-47.196,-180.000,4.288,148.697
C03658=1100.217,-117.532,-47.185,-180.000,4.283,148.695
C03659=1100.222,-117.781,-47.175,-179.998,4.278,148.694
C03660=1100.227,-118.030,-47.166,-179.998,4.273,148.693
C03661=1100.233,-118.281,-47.156,-179.997,4.267,148.691
C03662=1100.238,-118.531,-47.145,-179.997,4.262,148.690
C03663=1100.244,-118.780,-47.135,-179.996,4.258,148.689
C03664=1100.248,-119.030,-47.125,-179.995,4.252,148.687
C03665=1100.254,-119.280,-47.115,-179.995,4.247,148.686
C03666=1100.259,-119.529,-47.105,-179.994,4.242,148.685
C03667=1100.264,-119.779,-47.096,-179.994,4.236,148.683
C03668=1100.269,-120.029,-47.085,-179.993,4.232,148.682
C03669=1100.275,-120.279,-47.075,-179.992,4.226,148.681
C03670=1100.280,-120.528,-47.066,-179.992,4.221,148.680
C03671=1100.285,-120.778,-47.055,-179.991,4.216,148.678
C03672=1100.290,-121.028,-47.046,-179.991,4.211,148.677
C03673=1100.296,-121.278,-47.036,-179.990,4.205,148.675
C03674=1100.301,-121.527,-47.026,-179.989,4.201,148.674
C03675=1100.305,-121.777,-47.016,-179.988,4.195,148.673
C03676=1100.311,-122.027,-47.006,-179.988,4.190,148.672
C03677=1100.317,-122.277,-46.996,-179.988,4.185,148.670
C03678=1100.322,-122.526,-46.986,-179.987,4.179,148.669
